// TIA Portal V20 export
FUNCTION_BLOCK "Sequence_1_HotPressLeft"   // FB32858, LAD
TITLE = Sequence
// Sequence template programmend in ladder logic
// stored: IsIECCheckEnabled true, MemoryReserve 100, Namespace Unit1.Em6, SetENOAutomatically true
   VAR_INPUT
      unitStatus { ExternalAccessible := 'False'; ExternalVisible := 'False'; ExternalWritable := 'False'} : "LAF_typeUnitStatus";   // Current unit status o be used in this EM
   END_VAR
   VAR
      instSequenceLADControl { ExternalAccessible := 'False'; ExternalVisible := 'False'; ExternalWritable := 'False'} : "LAF_ControlLadSequence";
      instSequenceLADStatus { ExternalAccessible := 'False'; ExternalVisible := 'False'; ExternalWritable := 'False'} : "LAF_StatusLadSequence";
      statTonTime { ExternalAccessible := 'False'; ExternalVisible := 'False'; ExternalWritable := 'False'} : Array[0..9999] of TON_TIME;
      NoDataCheck { S7_SetPoint := 'True'} : "LER_typePartData";
   END_VAR
   VAR_TEMP
      tempCustomerAction : Bool;   // Placeholder for possible actions
      tempDo_nothing_and_wait_for_init : Bool;   // Placeholder for doing nothing
      tempSafeStateCondition : Bool;   // Temp Condition for the equipment module to be in a safe state
   END_VAR
   VAR CONSTANT
      delayTime : Time := T#500ms;
      STEP_IDLE : DInt := 1;
      JOB_1_STEP_01 : DInt := 101;
      JOB_1_STEP_10 : DInt := 110;
      JOB_1_STEP_20 : DInt := 120;
      JOB_1_STEP_30 : DInt := 130;
      JOB_1_STEP_40 : DInt := 140;
      JOB_1_STEP_41 : DInt := 141;
      JOB_1_STEP_50 : DInt := 150;
      JOB_1_STEP_60 : DInt := 160;
      JOB_1_STEP_70 : DInt := 170;
      JOB_1_STEP_80 : DInt := 180;
      JOB_1_STEP_90 : DInt := 190;
      JOB_2_STEP_01 : DInt := 201;
      JOB_2_STEP_10 : DInt := 210;
      JOB_2_STEP_20 : DInt := 220;
      JOB_2_STEP_30 : DInt := 230;
      JOB_2_STEP_31 : DInt := 231;
      JOB_2_STEP_32 : DInt := 232;
      JOB_2_STEP_40 : DInt := 240;
      JOB_2_STEP_41 : DInt := 241;
      JOB_2_STEP_42 : DInt := 242;
      JOB_2_STEP_43 : DInt := 242;
      JOB_2_STEP_50 : DInt := 250;
      JOB_2_STEP_60 : DInt := 260;
      JOB_2_STEP_70 : DInt := 270;
      JOB_2_STEP_80 : DInt := 280;
      JOB_2_STEP_90 : DInt := 290;
      JOB_3_STEP_01 : DInt := 301;
      JOB_3_STEP_10 : DInt := 310;
      JOB_3_STEP_11 : DInt := 311;
      JOB_3_STEP_20 : DInt := 320;
      JOB_3_STEP_30 : DInt := 330;
      JOB_3_STEP_31 : DInt := 331;
      JOB_3_STEP_32 : DInt := 332;
      JOB_3_STEP_33 : DInt := 333;
      JOB_3_STEP_40 : DInt := 340;
      JOB_3_STEP_41 : DInt := 341;
      JOB_3_STEP_42 : DInt := 342;
      JOB_3_STEP_43 : DInt := 343;
      JOB_3_STEP_50 : DInt := 350;
      JOB_3_STEP_60 : DInt := 360;
      JOB_3_STEP_70 : DInt := 370;
      JOB_3_STEP_80 : DInt := 380;
      JOB_3_STEP_90 : DInt := 390;
      JOB_4_STEP_01 : DInt := 401;
      JOB_4_STEP_10 : DInt := 410;
      JOB_4_STEP_20 : DInt := 420;
      JOB_4_STEP_30 : DInt := 430;
      JOB_4_STEP_31 : DInt := 431;
      JOB_4_STEP_40 : DInt := 440;
      JOB_4_STEP_41 : DInt := 441;
      JOB_4_STEP_42 : DInt := 442;
      JOB_4_STEP_50 : DInt := 450;
      JOB_4_STEP_60 : DInt := 460;
      JOB_4_STEP_70 : DInt := 470;
      JOB_4_STEP_80 : DInt := 480;
      JOB_4_STEP_81 : DInt := 481;
      JOB_4_STEP_90 : DInt := 490;
      JOB_5_STEP_01 : DInt := 501;
      JOB_5_STEP_10 : DInt := 510;
      JOB_5_STEP_11 : DInt := 511;
      JOB_5_STEP_12 : DInt := 512;
      JOB_5_STEP_13 : DInt := 513;
      JOB_5_STEP_20 : DInt := 520;
      JOB_5_STEP_30 : DInt := 530;
      JOB_5_STEP_40 : DInt := 540;
      JOB_5_STEP_41 : DInt := 541;
      JOB_5_STEP_42 : DInt := 542;
      JOB_5_STEP_50 : DInt := 550;
      JOB_5_STEP_60 : DInt := 560;
      JOB_5_STEP_61 : DInt := 561;
      JOB_5_STEP_62 : DInt := 562;
      JOB_5_STEP_63 : DInt := 563;
      JOB_5_STEP_64 : DInt := 564;
      JOB_5_STEP_70 : DInt := 570;
      JOB_5_STEP_80 : DInt := 580;
      JOB_5_STEP_90 : DInt := 590;
      STEP_IMMEDIATE_STOP : DInt := 9001;   // Step executed when an immediate stop command is triggered for the sequence (i.e. when unit is in state aborting)
   END_VAR
   VAR_TEMP   // added for the SCL form of the ladder/FBD networks
      _w1 : Bool;
   END_VAR
BEGIN

REGION Network 1: BLOCK INFO HEADER
   // (company) / (C) Copyright (year)
   // ---------------------------------------------------------------------------------
   // Title:                             (Title of this block)
   // Comment/Function: (that is implemented in the block)
   // Library/Family:           (that the source is dedicated to)
   // Author:                        (department / person in charge / contact)
   // Target System:          (test system with FW version)
   // Engineering:              TIA Portal (SW version)
   // Restrictions:               (OB types, etc.)
   // Requirements:           (hardware, technological package, etc.)
   // ---------------------------------------------------------------------------------
   // Change log table:
   // Version          | Date             | Signature      | Expert in charge  | Changes applied ------------------------|----------------------|-------------------------|--------------------------------|-----------------------
   // 001.000.000 | yyyy-mm-dd | 0x00000000 | (name of expert) | First released version
END_REGION

REGION Network 2: DESCRIPTION
   // This is a template block provided by the Automation Framework. It can be used to create an own project.
   // The Block Info Header is prepared to put in your own data.
   // Description of the block could be added here and the docu created by Code2Docu.
END_REGION

REGION Network 3: ********************* CONTROL *************************
END_REGION

REGION Network 4: Sequence Control ("Enter your Sequins number here")
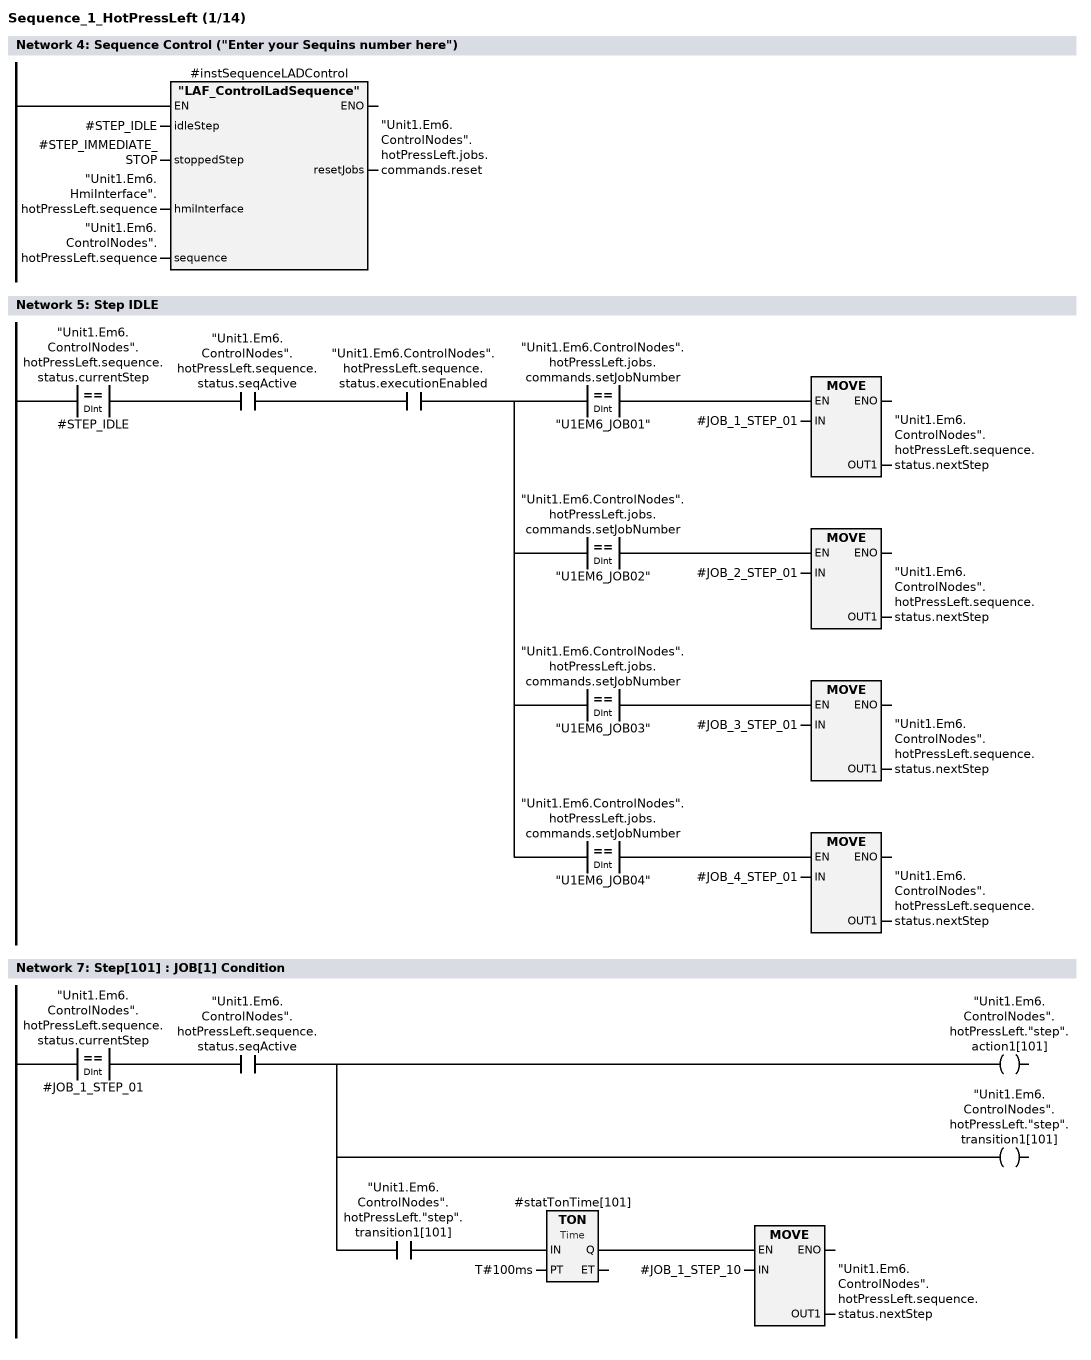
   RUNG wire#powerrail
      #instSequenceLADControl(idleStep := #STEP_IDLE, stoppedStep := #STEP_IMMEDIATE_STOP, hmiInterface := "Unit1.Em6.HmiInterface".hotPressLeft.sequence, sequence := "Unit1.Em6.ControlNodes".hotPressLeft.sequence, resetJobs => "Unit1.Em6.ControlNodes".hotPressLeft.jobs.commands.reset)
   END_RUNG
   // the same network as SCL:
   #instSequenceLADControl(idleStep := #STEP_IDLE,   // "LAF_ControlLadSequence"
                           stoppedStep := #STEP_IMMEDIATE_STOP,
                           hmiInterface := "Unit1.Em6.HmiInterface".hotPressLeft.sequence,
                           sequence := "Unit1.Em6.ControlNodes".hotPressLeft.sequence,
                           resetJobs => "Unit1.Em6.ControlNodes".hotPressLeft.jobs.commands.reset);
END_REGION

REGION Network 5: Step IDLE
   RUNG wire#powerrail
      { S7_Templates := "SrcType := DInt" } EQ_Contact(in1 := "Unit1.Em6.ControlNodes".hotPressLeft.sequence.status.currentStep, in2 := #STEP_IDLE)
      Contact( "Unit1.Em6.ControlNodes".hotPressLeft.sequence.status.seqActive )
      Contact( "Unit1.Em6.ControlNodes".hotPressLeft.sequence.status.executionEnabled )
      wire#w1
      { S7_Templates := "SrcType := DInt" } EQ_Contact(in1 := "Unit1.Em6.ControlNodes".hotPressLeft.jobs.commands.setJobNumber, in2 := "U1EM6_JOB01")
      Move(in := #JOB_1_STEP_01, out1 => "Unit1.Em6.ControlNodes".hotPressLeft.sequence.status.nextStep)
   END_RUNG
   RUNG wire#w1
      { S7_Templates := "SrcType := DInt" } EQ_Contact(in1 := "Unit1.Em6.ControlNodes".hotPressLeft.jobs.commands.setJobNumber, in2 := "U1EM6_JOB02")
      Move(in := #JOB_2_STEP_01, out1 => "Unit1.Em6.ControlNodes".hotPressLeft.sequence.status.nextStep)
   END_RUNG
   RUNG wire#w1
      { S7_Templates := "SrcType := DInt" } EQ_Contact(in1 := "Unit1.Em6.ControlNodes".hotPressLeft.jobs.commands.setJobNumber, in2 := "U1EM6_JOB03")
      Move(in := #JOB_3_STEP_01, out1 => "Unit1.Em6.ControlNodes".hotPressLeft.sequence.status.nextStep)
   END_RUNG
   RUNG wire#w1
      { S7_Templates := "SrcType := DInt" } EQ_Contact(in1 := "Unit1.Em6.ControlNodes".hotPressLeft.jobs.commands.setJobNumber, in2 := "U1EM6_JOB04")
      Move(in := #JOB_4_STEP_01, out1 => "Unit1.Em6.ControlNodes".hotPressLeft.sequence.status.nextStep)
   END_RUNG
   // the same network as SCL:
   #_w1 := ("Unit1.Em6.ControlNodes".hotPressLeft.sequence.status.currentStep = #STEP_IDLE) AND "Unit1.Em6.ControlNodes".hotPressLeft.sequence.status.seqActive AND "Unit1.Em6.ControlNodes".hotPressLeft.sequence.status.executionEnabled;
   IF #_w1 AND ("Unit1.Em6.ControlNodes".hotPressLeft.jobs.commands.setJobNumber = "U1EM6_JOB01") THEN
       "Unit1.Em6.ControlNodes".hotPressLeft.sequence.status.nextStep := #JOB_1_STEP_01;
   END_IF;
   IF #_w1 AND ("Unit1.Em6.ControlNodes".hotPressLeft.jobs.commands.setJobNumber = "U1EM6_JOB02") THEN
       "Unit1.Em6.ControlNodes".hotPressLeft.sequence.status.nextStep := #JOB_2_STEP_01;
   END_IF;
   IF #_w1 AND ("Unit1.Em6.ControlNodes".hotPressLeft.jobs.commands.setJobNumber = "U1EM6_JOB03") THEN
       "Unit1.Em6.ControlNodes".hotPressLeft.sequence.status.nextStep := #JOB_3_STEP_01;
   END_IF;
   IF #_w1 AND ("Unit1.Em6.ControlNodes".hotPressLeft.jobs.commands.setJobNumber = "U1EM6_JOB04") THEN
       "Unit1.Em6.ControlNodes".hotPressLeft.sequence.status.nextStep := #JOB_4_STEP_01;
   END_IF;
END_REGION

REGION Network 6: *************** JOB[1] EM HOMING ************************
END_REGION

REGION Network 7: Step[101] : JOB[1] Condition
   RUNG wire#powerrail
      { S7_Templates := "SrcType := DInt" } EQ_Contact(in1 := "Unit1.Em6.ControlNodes".hotPressLeft.sequence.status.currentStep, in2 := #JOB_1_STEP_01)
      Contact( "Unit1.Em6.ControlNodes".hotPressLeft.sequence.status.seqActive )
      wire#w1
      Coil( "Unit1.Em6.ControlNodes".hotPressLeft."step".action1[101] )
   END_RUNG
   RUNG wire#w1
      Coil( "Unit1.Em6.ControlNodes".hotPressLeft."step".transition1[101] )
   END_RUNG
   RUNG wire#w1
      Contact( "Unit1.Em6.ControlNodes".hotPressLeft."step".transition1[101] )
      { S7_Templates := "time_type := Time" } #statTonTime[101].TON(pt := T#100ms, et =>)
      Move(in := #JOB_1_STEP_10, out1 => "Unit1.Em6.ControlNodes".hotPressLeft.sequence.status.nextStep)
   END_RUNG
   // the same network as SCL:
   "Unit1.Em6.ControlNodes".hotPressLeft."step".action1[101] := ("Unit1.Em6.ControlNodes".hotPressLeft.sequence.status.currentStep = #JOB_1_STEP_01) AND "Unit1.Em6.ControlNodes".hotPressLeft.sequence.status.seqActive;
   "Unit1.Em6.ControlNodes".hotPressLeft."step".transition1[101] := ("Unit1.Em6.ControlNodes".hotPressLeft.sequence.status.currentStep = #JOB_1_STEP_01) AND "Unit1.Em6.ControlNodes".hotPressLeft.sequence.status.seqActive;
   #statTonTime[101].TON(IN := ("Unit1.Em6.ControlNodes".hotPressLeft.sequence.status.currentStep = #JOB_1_STEP_01) AND "Unit1.Em6.ControlNodes".hotPressLeft.sequence.status.seqActive AND "Unit1.Em6.ControlNodes".hotPressLeft."step".transition1[101],
                         PT := T#100ms);
   IF #statTonTime[101].Q THEN
       "Unit1.Em6.ControlNodes".hotPressLeft.sequence.status.nextStep := #JOB_1_STEP_10;
   END_IF;
END_REGION

REGION Network 8: Step[110] : Servo Press Reference Home Pos
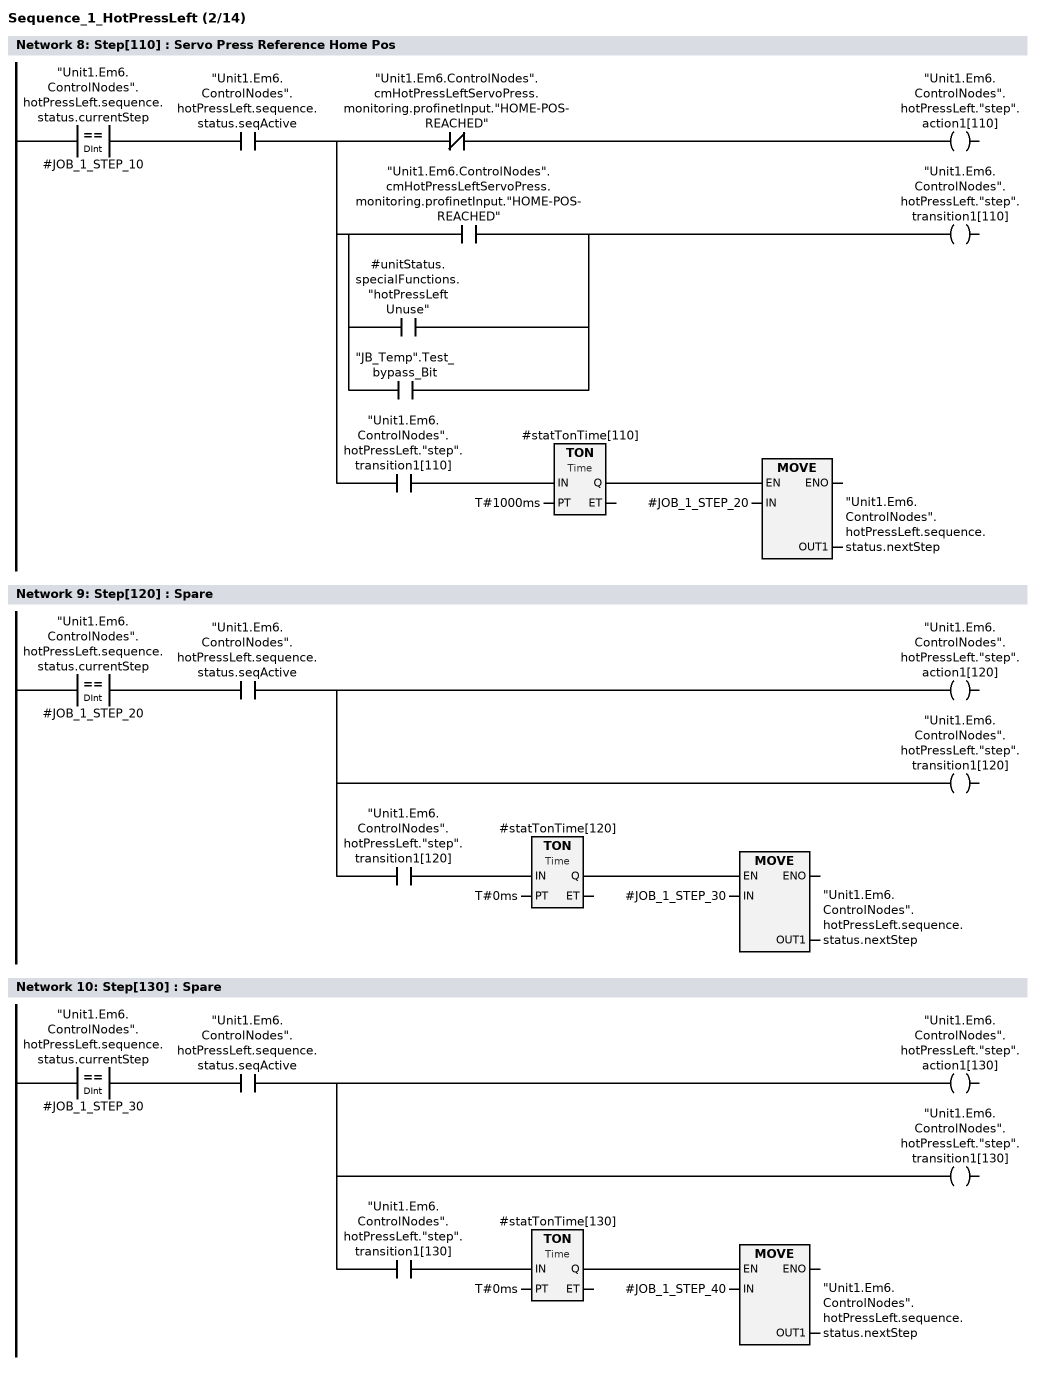
   RUNG wire#powerrail
      { S7_Templates := "SrcType := DInt" } EQ_Contact(in1 := "Unit1.Em6.ControlNodes".hotPressLeft.sequence.status.currentStep, in2 := #JOB_1_STEP_10)
      Contact( "Unit1.Em6.ControlNodes".hotPressLeft.sequence.status.seqActive )
      wire#w1
      I_Contact( "Unit1.Em6.ControlNodes".cmHotPressLeftServoPress.monitoring.profinetInput."HOME-POS-REACHED" )
      Coil( "Unit1.Em6.ControlNodes".hotPressLeft."step".action1[110] )
   END_RUNG
   RUNG wire#w1
      Contact( "Unit1.Em6.ControlNodes".cmHotPressLeftServoPress.monitoring.profinetInput."HOME-POS-REACHED" )
      wire#w2
      Coil( "Unit1.Em6.ControlNodes".hotPressLeft."step".transition1[110] )
   END_RUNG
   RUNG wire#w1
      Contact( #unitStatus.specialFunctions."hotPressLeft Unuse" )
   END_RUNG wire#w2
   RUNG wire#w1
      Contact( "JB_Temp".Test_bypass_Bit )
   END_RUNG wire#w2
   RUNG wire#w1
      Contact( "Unit1.Em6.ControlNodes".hotPressLeft."step".transition1[110] )
      { S7_Templates := "time_type := Time" } #statTonTime[110].TON(pt := T#1000ms, et =>)
      Move(in := #JOB_1_STEP_20, out1 => "Unit1.Em6.ControlNodes".hotPressLeft.sequence.status.nextStep)
   END_RUNG
   // the same network as SCL:
   #_w1 := ("Unit1.Em6.ControlNodes".hotPressLeft.sequence.status.currentStep = #JOB_1_STEP_10) AND "Unit1.Em6.ControlNodes".hotPressLeft.sequence.status.seqActive;
   "Unit1.Em6.ControlNodes".hotPressLeft."step".action1[110] := #_w1 AND NOT "Unit1.Em6.ControlNodes".cmHotPressLeftServoPress.monitoring.profinetInput."HOME-POS-REACHED";
   "Unit1.Em6.ControlNodes".hotPressLeft."step".transition1[110] := #_w1 AND ("Unit1.Em6.ControlNodes".cmHotPressLeftServoPress.monitoring.profinetInput."HOME-POS-REACHED" OR #unitStatus.specialFunctions."hotPressLeft Unuse" OR "JB_Temp".Test_bypass_Bit);
   #statTonTime[110].TON(IN := #_w1 AND "Unit1.Em6.ControlNodes".hotPressLeft."step".transition1[110],
                         PT := T#1000ms);
   IF #statTonTime[110].Q THEN
       "Unit1.Em6.ControlNodes".hotPressLeft.sequence.status.nextStep := #JOB_1_STEP_20;
   END_IF;
END_REGION

REGION Network 9: Step[120] : Spare
   RUNG wire#powerrail
      { S7_Templates := "SrcType := DInt" } EQ_Contact(in1 := "Unit1.Em6.ControlNodes".hotPressLeft.sequence.status.currentStep, in2 := #JOB_1_STEP_20)
      Contact( "Unit1.Em6.ControlNodes".hotPressLeft.sequence.status.seqActive )
      wire#w1
      Coil( "Unit1.Em6.ControlNodes".hotPressLeft."step".action1[120] )
   END_RUNG
   RUNG wire#w1
      Coil( "Unit1.Em6.ControlNodes".hotPressLeft."step".transition1[120] )
   END_RUNG
   RUNG wire#w1
      Contact( "Unit1.Em6.ControlNodes".hotPressLeft."step".transition1[120] )
      { S7_Templates := "time_type := Time" } #statTonTime[120].TON(pt := T#0ms, et =>)
      Move(in := #JOB_1_STEP_30, out1 => "Unit1.Em6.ControlNodes".hotPressLeft.sequence.status.nextStep)
   END_RUNG
   // the same network as SCL:
   "Unit1.Em6.ControlNodes".hotPressLeft."step".action1[120] := ("Unit1.Em6.ControlNodes".hotPressLeft.sequence.status.currentStep = #JOB_1_STEP_20) AND "Unit1.Em6.ControlNodes".hotPressLeft.sequence.status.seqActive;
   "Unit1.Em6.ControlNodes".hotPressLeft."step".transition1[120] := ("Unit1.Em6.ControlNodes".hotPressLeft.sequence.status.currentStep = #JOB_1_STEP_20) AND "Unit1.Em6.ControlNodes".hotPressLeft.sequence.status.seqActive;
   #statTonTime[120].TON(IN := ("Unit1.Em6.ControlNodes".hotPressLeft.sequence.status.currentStep = #JOB_1_STEP_20) AND "Unit1.Em6.ControlNodes".hotPressLeft.sequence.status.seqActive AND "Unit1.Em6.ControlNodes".hotPressLeft."step".transition1[120],
                         PT := T#0ms);
   IF #statTonTime[120].Q THEN
       "Unit1.Em6.ControlNodes".hotPressLeft.sequence.status.nextStep := #JOB_1_STEP_30;
   END_IF;
END_REGION

REGION Network 10: Step[130] : Spare
   RUNG wire#powerrail
      { S7_Templates := "SrcType := DInt" } EQ_Contact(in1 := "Unit1.Em6.ControlNodes".hotPressLeft.sequence.status.currentStep, in2 := #JOB_1_STEP_30)
      Contact( "Unit1.Em6.ControlNodes".hotPressLeft.sequence.status.seqActive )
      wire#w1
      Coil( "Unit1.Em6.ControlNodes".hotPressLeft."step".action1[130] )
   END_RUNG
   RUNG wire#w1
      Coil( "Unit1.Em6.ControlNodes".hotPressLeft."step".transition1[130] )
   END_RUNG
   RUNG wire#w1
      Contact( "Unit1.Em6.ControlNodes".hotPressLeft."step".transition1[130] )
      { S7_Templates := "time_type := Time" } #statTonTime[130].TON(pt := T#0ms, et =>)
      Move(in := #JOB_1_STEP_40, out1 => "Unit1.Em6.ControlNodes".hotPressLeft.sequence.status.nextStep)
   END_RUNG
   // the same network as SCL:
   "Unit1.Em6.ControlNodes".hotPressLeft."step".action1[130] := ("Unit1.Em6.ControlNodes".hotPressLeft.sequence.status.currentStep = #JOB_1_STEP_30) AND "Unit1.Em6.ControlNodes".hotPressLeft.sequence.status.seqActive;
   "Unit1.Em6.ControlNodes".hotPressLeft."step".transition1[130] := ("Unit1.Em6.ControlNodes".hotPressLeft.sequence.status.currentStep = #JOB_1_STEP_30) AND "Unit1.Em6.ControlNodes".hotPressLeft.sequence.status.seqActive;
   #statTonTime[130].TON(IN := ("Unit1.Em6.ControlNodes".hotPressLeft.sequence.status.currentStep = #JOB_1_STEP_30) AND "Unit1.Em6.ControlNodes".hotPressLeft.sequence.status.seqActive AND "Unit1.Em6.ControlNodes".hotPressLeft."step".transition1[130],
                         PT := T#0ms);
   IF #statTonTime[130].Q THEN
       "Unit1.Em6.ControlNodes".hotPressLeft.sequence.status.nextStep := #JOB_1_STEP_40;
   END_IF;
END_REGION

REGION Network 11: Step[140] : Spare
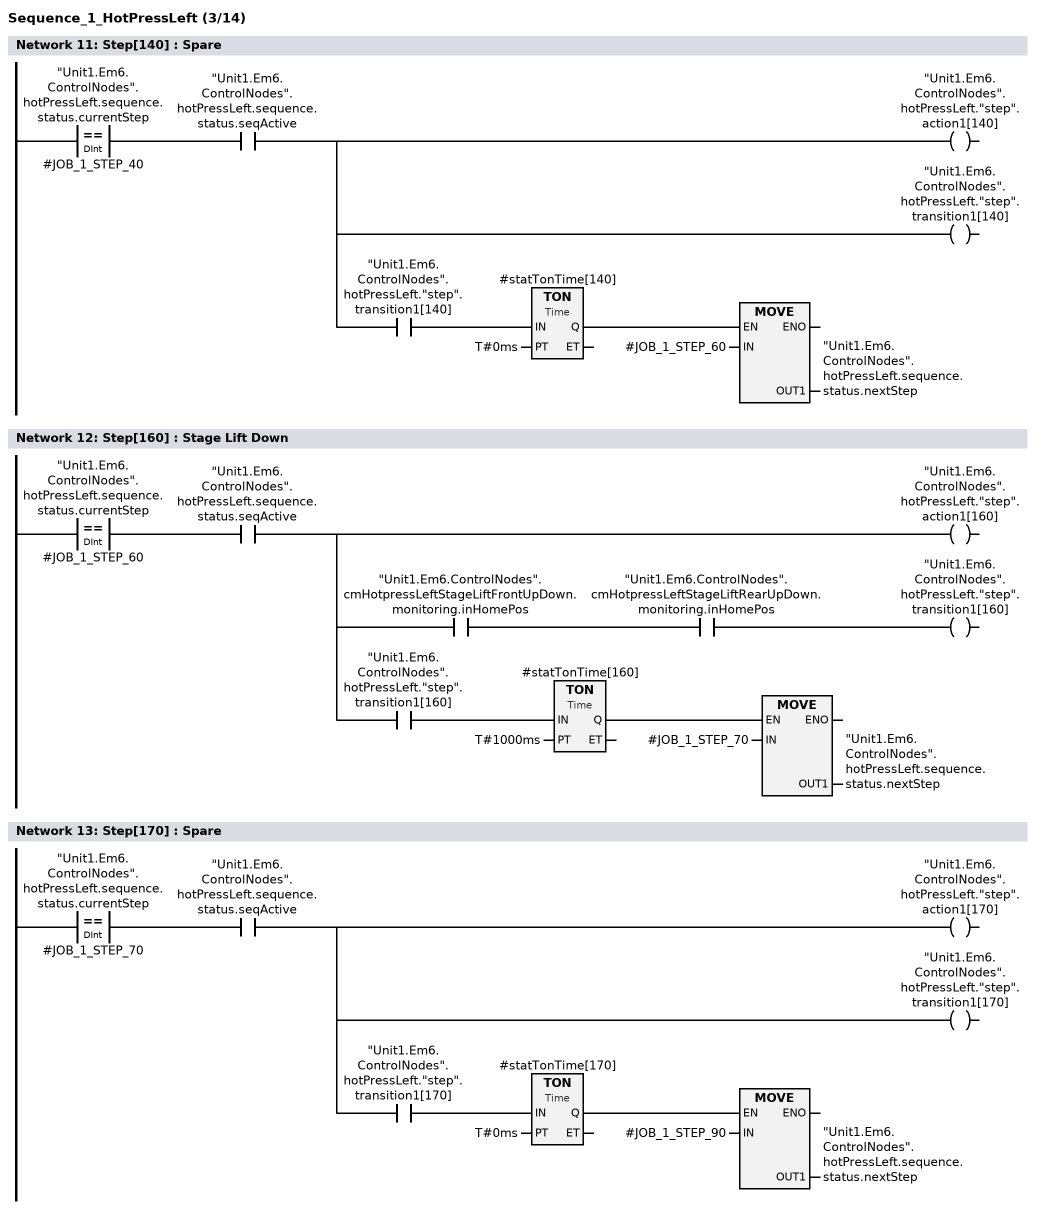
   RUNG wire#powerrail
      { S7_Templates := "SrcType := DInt" } EQ_Contact(in1 := "Unit1.Em6.ControlNodes".hotPressLeft.sequence.status.currentStep, in2 := #JOB_1_STEP_40)
      Contact( "Unit1.Em6.ControlNodes".hotPressLeft.sequence.status.seqActive )
      wire#w1
      Coil( "Unit1.Em6.ControlNodes".hotPressLeft."step".action1[140] )
   END_RUNG
   RUNG wire#w1
      Coil( "Unit1.Em6.ControlNodes".hotPressLeft."step".transition1[140] )
   END_RUNG
   RUNG wire#w1
      Contact( "Unit1.Em6.ControlNodes".hotPressLeft."step".transition1[140] )
      { S7_Templates := "time_type := Time" } #statTonTime[140].TON(pt := T#0ms, et =>)
      Move(in := #JOB_1_STEP_60, out1 => "Unit1.Em6.ControlNodes".hotPressLeft.sequence.status.nextStep)
   END_RUNG
   // the same network as SCL:
   "Unit1.Em6.ControlNodes".hotPressLeft."step".action1[140] := ("Unit1.Em6.ControlNodes".hotPressLeft.sequence.status.currentStep = #JOB_1_STEP_40) AND "Unit1.Em6.ControlNodes".hotPressLeft.sequence.status.seqActive;
   "Unit1.Em6.ControlNodes".hotPressLeft."step".transition1[140] := ("Unit1.Em6.ControlNodes".hotPressLeft.sequence.status.currentStep = #JOB_1_STEP_40) AND "Unit1.Em6.ControlNodes".hotPressLeft.sequence.status.seqActive;
   #statTonTime[140].TON(IN := ("Unit1.Em6.ControlNodes".hotPressLeft.sequence.status.currentStep = #JOB_1_STEP_40) AND "Unit1.Em6.ControlNodes".hotPressLeft.sequence.status.seqActive AND "Unit1.Em6.ControlNodes".hotPressLeft."step".transition1[140],
                         PT := T#0ms);
   IF #statTonTime[140].Q THEN
       "Unit1.Em6.ControlNodes".hotPressLeft.sequence.status.nextStep := #JOB_1_STEP_60;
   END_IF;
END_REGION

REGION Network 12: Step[160] : Stage Lift Down
   RUNG wire#powerrail
      { S7_Templates := "SrcType := DInt" } EQ_Contact(in1 := "Unit1.Em6.ControlNodes".hotPressLeft.sequence.status.currentStep, in2 := #JOB_1_STEP_60)
      Contact( "Unit1.Em6.ControlNodes".hotPressLeft.sequence.status.seqActive )
      wire#w1
      Coil( "Unit1.Em6.ControlNodes".hotPressLeft."step".action1[160] )
   END_RUNG
   RUNG wire#w1
      Contact( "Unit1.Em6.ControlNodes".cmHotpressLeftStageLiftFrontUpDown.monitoring.inHomePos )
      Contact( "Unit1.Em6.ControlNodes".cmHotpressLeftStageLiftRearUpDown.monitoring.inHomePos )
      Coil( "Unit1.Em6.ControlNodes".hotPressLeft."step".transition1[160] )
   END_RUNG
   RUNG wire#w1
      Contact( "Unit1.Em6.ControlNodes".hotPressLeft."step".transition1[160] )
      { S7_Templates := "time_type := Time" } #statTonTime[160].TON(pt := T#1000ms, et =>)
      Move(in := #JOB_1_STEP_70, out1 => "Unit1.Em6.ControlNodes".hotPressLeft.sequence.status.nextStep)
   END_RUNG
   // the same network as SCL:
   "Unit1.Em6.ControlNodes".hotPressLeft."step".action1[160] := ("Unit1.Em6.ControlNodes".hotPressLeft.sequence.status.currentStep = #JOB_1_STEP_60) AND "Unit1.Em6.ControlNodes".hotPressLeft.sequence.status.seqActive;
   "Unit1.Em6.ControlNodes".hotPressLeft."step".transition1[160] := ("Unit1.Em6.ControlNodes".hotPressLeft.sequence.status.currentStep = #JOB_1_STEP_60) AND "Unit1.Em6.ControlNodes".hotPressLeft.sequence.status.seqActive AND "Unit1.Em6.ControlNodes".cmHotpressLeftStageLiftFrontUpDown.monitoring.inHomePos AND "Unit1.Em6.ControlNodes".cmHotpressLeftStageLiftRearUpDown.monitoring.inHomePos;
   #statTonTime[160].TON(IN := ("Unit1.Em6.ControlNodes".hotPressLeft.sequence.status.currentStep = #JOB_1_STEP_60) AND "Unit1.Em6.ControlNodes".hotPressLeft.sequence.status.seqActive AND "Unit1.Em6.ControlNodes".hotPressLeft."step".transition1[160],
                         PT := T#1000ms);
   IF #statTonTime[160].Q THEN
       "Unit1.Em6.ControlNodes".hotPressLeft.sequence.status.nextStep := #JOB_1_STEP_70;
   END_IF;
END_REGION

REGION Network 13: Step[170] : Spare
   RUNG wire#powerrail
      { S7_Templates := "SrcType := DInt" } EQ_Contact(in1 := "Unit1.Em6.ControlNodes".hotPressLeft.sequence.status.currentStep, in2 := #JOB_1_STEP_70)
      Contact( "Unit1.Em6.ControlNodes".hotPressLeft.sequence.status.seqActive )
      wire#w1
      Coil( "Unit1.Em6.ControlNodes".hotPressLeft."step".action1[170] )
   END_RUNG
   RUNG wire#w1
      Coil( "Unit1.Em6.ControlNodes".hotPressLeft."step".transition1[170] )
   END_RUNG
   RUNG wire#w1
      Contact( "Unit1.Em6.ControlNodes".hotPressLeft."step".transition1[170] )
      { S7_Templates := "time_type := Time" } #statTonTime[170].TON(pt := T#0ms, et =>)
      Move(in := #JOB_1_STEP_90, out1 => "Unit1.Em6.ControlNodes".hotPressLeft.sequence.status.nextStep)
   END_RUNG
   // the same network as SCL:
   "Unit1.Em6.ControlNodes".hotPressLeft."step".action1[170] := ("Unit1.Em6.ControlNodes".hotPressLeft.sequence.status.currentStep = #JOB_1_STEP_70) AND "Unit1.Em6.ControlNodes".hotPressLeft.sequence.status.seqActive;
   "Unit1.Em6.ControlNodes".hotPressLeft."step".transition1[170] := ("Unit1.Em6.ControlNodes".hotPressLeft.sequence.status.currentStep = #JOB_1_STEP_70) AND "Unit1.Em6.ControlNodes".hotPressLeft.sequence.status.seqActive;
   #statTonTime[170].TON(IN := ("Unit1.Em6.ControlNodes".hotPressLeft.sequence.status.currentStep = #JOB_1_STEP_70) AND "Unit1.Em6.ControlNodes".hotPressLeft.sequence.status.seqActive AND "Unit1.Em6.ControlNodes".hotPressLeft."step".transition1[170],
                         PT := T#0ms);
   IF #statTonTime[170].Q THEN
       "Unit1.Em6.ControlNodes".hotPressLeft.sequence.status.nextStep := #JOB_1_STEP_90;
   END_IF;
END_REGION

REGION Network 14: Step[190] : JOB[1] Step End
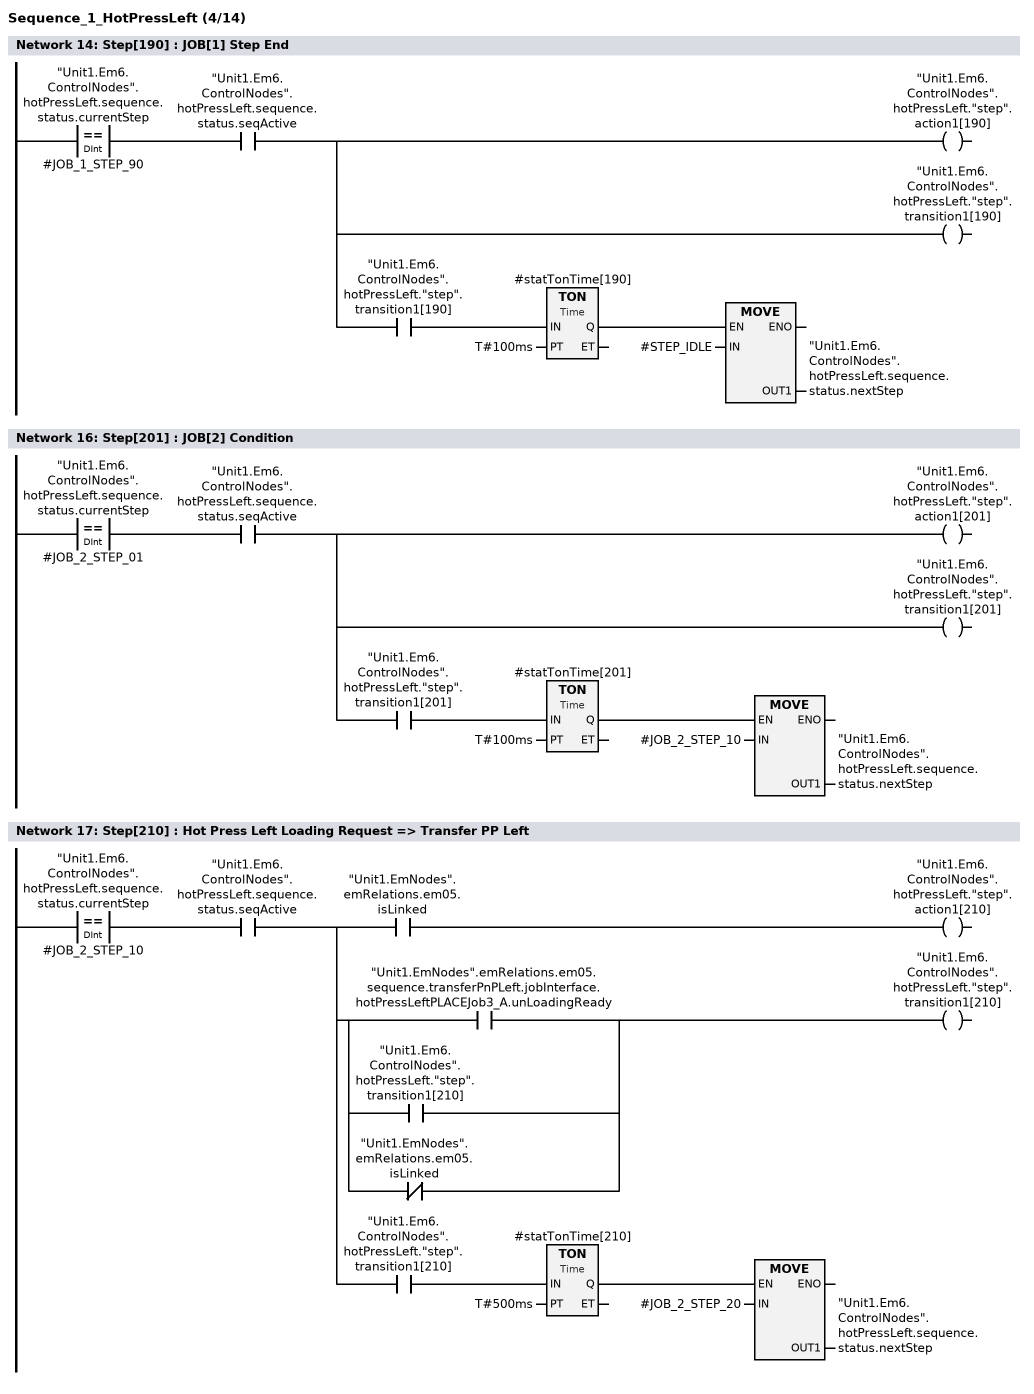
   RUNG wire#powerrail
      { S7_Templates := "SrcType := DInt" } EQ_Contact(in1 := "Unit1.Em6.ControlNodes".hotPressLeft.sequence.status.currentStep, in2 := #JOB_1_STEP_90)
      Contact( "Unit1.Em6.ControlNodes".hotPressLeft.sequence.status.seqActive )
      wire#w1
      Coil( "Unit1.Em6.ControlNodes".hotPressLeft."step".action1[190] )
   END_RUNG
   RUNG wire#w1
      Coil( "Unit1.Em6.ControlNodes".hotPressLeft."step".transition1[190] )
   END_RUNG
   RUNG wire#w1
      Contact( "Unit1.Em6.ControlNodes".hotPressLeft."step".transition1[190] )
      { S7_Templates := "time_type := Time" } #statTonTime[190].TON(pt := T#100ms, et =>)
      Move(in := #STEP_IDLE, out1 => "Unit1.Em6.ControlNodes".hotPressLeft.sequence.status.nextStep)
   END_RUNG
   // the same network as SCL:
   "Unit1.Em6.ControlNodes".hotPressLeft."step".action1[190] := ("Unit1.Em6.ControlNodes".hotPressLeft.sequence.status.currentStep = #JOB_1_STEP_90) AND "Unit1.Em6.ControlNodes".hotPressLeft.sequence.status.seqActive;
   "Unit1.Em6.ControlNodes".hotPressLeft."step".transition1[190] := ("Unit1.Em6.ControlNodes".hotPressLeft.sequence.status.currentStep = #JOB_1_STEP_90) AND "Unit1.Em6.ControlNodes".hotPressLeft.sequence.status.seqActive;
   #statTonTime[190].TON(IN := ("Unit1.Em6.ControlNodes".hotPressLeft.sequence.status.currentStep = #JOB_1_STEP_90) AND "Unit1.Em6.ControlNodes".hotPressLeft.sequence.status.seqActive AND "Unit1.Em6.ControlNodes".hotPressLeft."step".transition1[190],
                         PT := T#100ms);
   IF #statTonTime[190].Q THEN
       "Unit1.Em6.ControlNodes".hotPressLeft.sequence.status.nextStep := #STEP_IDLE;
   END_IF;
END_REGION

REGION Network 15: *************** JOB[2] JR GET=AUTO **********************
END_REGION

REGION Network 16: Step[201] : JOB[2] Condition
   RUNG wire#powerrail
      { S7_Templates := "SrcType := DInt" } EQ_Contact(in1 := "Unit1.Em6.ControlNodes".hotPressLeft.sequence.status.currentStep, in2 := #JOB_2_STEP_01)
      Contact( "Unit1.Em6.ControlNodes".hotPressLeft.sequence.status.seqActive )
      wire#w1
      Coil( "Unit1.Em6.ControlNodes".hotPressLeft."step".action1[201] )
   END_RUNG
   RUNG wire#w1
      Coil( "Unit1.Em6.ControlNodes".hotPressLeft."step".transition1[201] )
   END_RUNG
   RUNG wire#w1
      Contact( "Unit1.Em6.ControlNodes".hotPressLeft."step".transition1[201] )
      { S7_Templates := "time_type := Time" } #statTonTime[201].TON(pt := T#100ms, et =>)
      Move(in := #JOB_2_STEP_10, out1 => "Unit1.Em6.ControlNodes".hotPressLeft.sequence.status.nextStep)
   END_RUNG
   // the same network as SCL:
   "Unit1.Em6.ControlNodes".hotPressLeft."step".action1[201] := ("Unit1.Em6.ControlNodes".hotPressLeft.sequence.status.currentStep = #JOB_2_STEP_01) AND "Unit1.Em6.ControlNodes".hotPressLeft.sequence.status.seqActive;
   "Unit1.Em6.ControlNodes".hotPressLeft."step".transition1[201] := ("Unit1.Em6.ControlNodes".hotPressLeft.sequence.status.currentStep = #JOB_2_STEP_01) AND "Unit1.Em6.ControlNodes".hotPressLeft.sequence.status.seqActive;
   #statTonTime[201].TON(IN := ("Unit1.Em6.ControlNodes".hotPressLeft.sequence.status.currentStep = #JOB_2_STEP_01) AND "Unit1.Em6.ControlNodes".hotPressLeft.sequence.status.seqActive AND "Unit1.Em6.ControlNodes".hotPressLeft."step".transition1[201],
                         PT := T#100ms);
   IF #statTonTime[201].Q THEN
       "Unit1.Em6.ControlNodes".hotPressLeft.sequence.status.nextStep := #JOB_2_STEP_10;
   END_IF;
END_REGION

REGION Network 17: Step[210] : Hot Press Left Loading Request => Transfer PP Left
   RUNG wire#powerrail
      { S7_Templates := "SrcType := DInt" } EQ_Contact(in1 := "Unit1.Em6.ControlNodes".hotPressLeft.sequence.status.currentStep, in2 := #JOB_2_STEP_10)
      Contact( "Unit1.Em6.ControlNodes".hotPressLeft.sequence.status.seqActive )
      wire#w1
      Contact( "Unit1.EmNodes".emRelations.em05.isLinked )
      Coil( "Unit1.Em6.ControlNodes".hotPressLeft."step".action1[210] )
   END_RUNG
   RUNG wire#w1
      Contact( "Unit1.EmNodes".emRelations.em05.sequence.transferPnPLeft.jobInterface.hotPressLeftPLACEJob3_A.unLoadingReady )
      wire#w2
      Coil( "Unit1.Em6.ControlNodes".hotPressLeft."step".transition1[210] )
   END_RUNG
   RUNG wire#w1
      Contact( "Unit1.Em6.ControlNodes".hotPressLeft."step".transition1[210] )
   END_RUNG wire#w2
   RUNG wire#w1
      I_Contact( "Unit1.EmNodes".emRelations.em05.isLinked )
   END_RUNG wire#w2
   RUNG wire#w1
      Contact( "Unit1.Em6.ControlNodes".hotPressLeft."step".transition1[210] )
      { S7_Templates := "time_type := Time" } #statTonTime[210].TON(pt := T#500ms, et =>)
      Move(in := #JOB_2_STEP_20, out1 => "Unit1.Em6.ControlNodes".hotPressLeft.sequence.status.nextStep)
   END_RUNG
   // the same network as SCL:
   #_w1 := ("Unit1.Em6.ControlNodes".hotPressLeft.sequence.status.currentStep = #JOB_2_STEP_10) AND "Unit1.Em6.ControlNodes".hotPressLeft.sequence.status.seqActive;
   "Unit1.Em6.ControlNodes".hotPressLeft."step".action1[210] := #_w1 AND "Unit1.EmNodes".emRelations.em05.isLinked;
   "Unit1.Em6.ControlNodes".hotPressLeft."step".transition1[210] := #_w1 AND ("Unit1.EmNodes".emRelations.em05.sequence.transferPnPLeft.jobInterface.hotPressLeftPLACEJob3_A.unLoadingReady OR "Unit1.Em6.ControlNodes".hotPressLeft."step".transition1[210] OR NOT "Unit1.EmNodes".emRelations.em05.isLinked);
   #statTonTime[210].TON(IN := #_w1 AND "Unit1.Em6.ControlNodes".hotPressLeft."step".transition1[210],
                         PT := T#500ms);
   IF #statTonTime[210].Q THEN
       "Unit1.Em6.ControlNodes".hotPressLeft.sequence.status.nextStep := #JOB_2_STEP_20;
   END_IF;
END_REGION

REGION Network 18: Step[220] : Spare
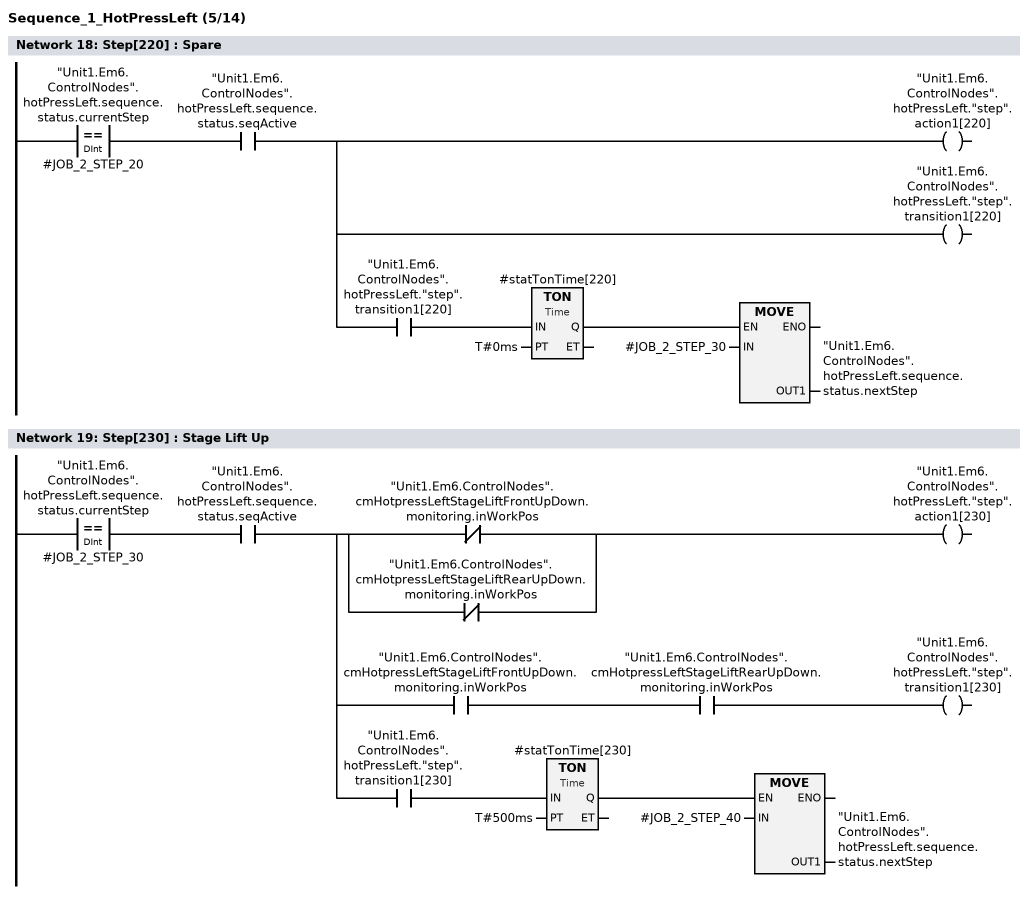
   RUNG wire#powerrail
      { S7_Templates := "SrcType := DInt" } EQ_Contact(in1 := "Unit1.Em6.ControlNodes".hotPressLeft.sequence.status.currentStep, in2 := #JOB_2_STEP_20)
      Contact( "Unit1.Em6.ControlNodes".hotPressLeft.sequence.status.seqActive )
      wire#w1
      Coil( "Unit1.Em6.ControlNodes".hotPressLeft."step".action1[220] )
   END_RUNG
   RUNG wire#w1
      Coil( "Unit1.Em6.ControlNodes".hotPressLeft."step".transition1[220] )
   END_RUNG
   RUNG wire#w1
      Contact( "Unit1.Em6.ControlNodes".hotPressLeft."step".transition1[220] )
      { S7_Templates := "time_type := Time" } #statTonTime[220].TON(pt := T#0ms, et =>)
      Move(in := #JOB_2_STEP_30, out1 => "Unit1.Em6.ControlNodes".hotPressLeft.sequence.status.nextStep)
   END_RUNG
   // the same network as SCL:
   "Unit1.Em6.ControlNodes".hotPressLeft."step".action1[220] := ("Unit1.Em6.ControlNodes".hotPressLeft.sequence.status.currentStep = #JOB_2_STEP_20) AND "Unit1.Em6.ControlNodes".hotPressLeft.sequence.status.seqActive;
   "Unit1.Em6.ControlNodes".hotPressLeft."step".transition1[220] := ("Unit1.Em6.ControlNodes".hotPressLeft.sequence.status.currentStep = #JOB_2_STEP_20) AND "Unit1.Em6.ControlNodes".hotPressLeft.sequence.status.seqActive;
   #statTonTime[220].TON(IN := ("Unit1.Em6.ControlNodes".hotPressLeft.sequence.status.currentStep = #JOB_2_STEP_20) AND "Unit1.Em6.ControlNodes".hotPressLeft.sequence.status.seqActive AND "Unit1.Em6.ControlNodes".hotPressLeft."step".transition1[220],
                         PT := T#0ms);
   IF #statTonTime[220].Q THEN
       "Unit1.Em6.ControlNodes".hotPressLeft.sequence.status.nextStep := #JOB_2_STEP_30;
   END_IF;
END_REGION

REGION Network 19: Step[230] : Stage Lift Up
   RUNG wire#powerrail
      { S7_Templates := "SrcType := DInt" } EQ_Contact(in1 := "Unit1.Em6.ControlNodes".hotPressLeft.sequence.status.currentStep, in2 := #JOB_2_STEP_30)
      Contact( "Unit1.Em6.ControlNodes".hotPressLeft.sequence.status.seqActive )
      wire#w1
      I_Contact( "Unit1.Em6.ControlNodes".cmHotpressLeftStageLiftFrontUpDown.monitoring.inWorkPos )
      wire#w2
      Coil( "Unit1.Em6.ControlNodes".hotPressLeft."step".action1[230] )
   END_RUNG
   RUNG wire#w1
      I_Contact( "Unit1.Em6.ControlNodes".cmHotpressLeftStageLiftRearUpDown.monitoring.inWorkPos )
   END_RUNG wire#w2
   RUNG wire#w1
      Contact( "Unit1.Em6.ControlNodes".cmHotpressLeftStageLiftFrontUpDown.monitoring.inWorkPos )
      Contact( "Unit1.Em6.ControlNodes".cmHotpressLeftStageLiftRearUpDown.monitoring.inWorkPos )
      Coil( "Unit1.Em6.ControlNodes".hotPressLeft."step".transition1[230] )
   END_RUNG
   RUNG wire#w1
      Contact( "Unit1.Em6.ControlNodes".hotPressLeft."step".transition1[230] )
      { S7_Templates := "time_type := Time" } #statTonTime[230].TON(pt := T#500ms, et =>)
      Move(in := #JOB_2_STEP_40, out1 => "Unit1.Em6.ControlNodes".hotPressLeft.sequence.status.nextStep)
   END_RUNG
   // the same network as SCL:
   #_w1 := ("Unit1.Em6.ControlNodes".hotPressLeft.sequence.status.currentStep = #JOB_2_STEP_30) AND "Unit1.Em6.ControlNodes".hotPressLeft.sequence.status.seqActive;
   "Unit1.Em6.ControlNodes".hotPressLeft."step".action1[230] := #_w1 AND (NOT "Unit1.Em6.ControlNodes".cmHotpressLeftStageLiftFrontUpDown.monitoring.inWorkPos OR NOT "Unit1.Em6.ControlNodes".cmHotpressLeftStageLiftRearUpDown.monitoring.inWorkPos);
   "Unit1.Em6.ControlNodes".hotPressLeft."step".transition1[230] := #_w1 AND "Unit1.Em6.ControlNodes".cmHotpressLeftStageLiftFrontUpDown.monitoring.inWorkPos AND "Unit1.Em6.ControlNodes".cmHotpressLeftStageLiftRearUpDown.monitoring.inWorkPos;
   #statTonTime[230].TON(IN := #_w1 AND "Unit1.Em6.ControlNodes".hotPressLeft."step".transition1[230],
                         PT := T#500ms);
   IF #statTonTime[230].Q THEN
       "Unit1.Em6.ControlNodes".hotPressLeft.sequence.status.nextStep := #JOB_2_STEP_40;
   END_IF;
END_REGION

REGION Network 20: Step[240] : Hot Press Left Loading Check => Transfer PP Left
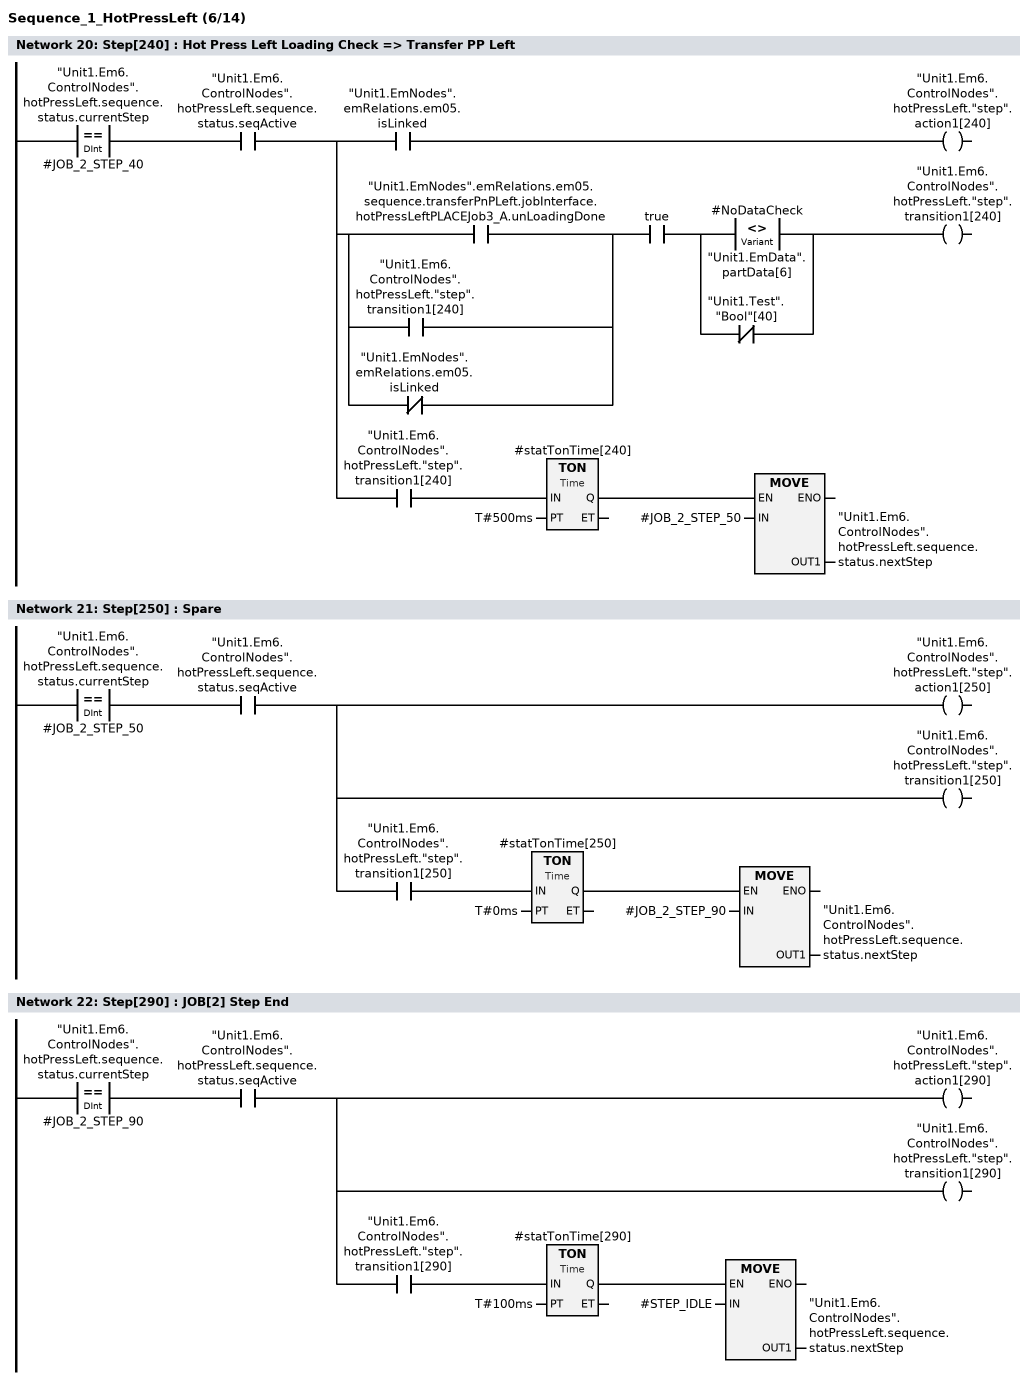
   RUNG wire#powerrail
      { S7_Templates := "SrcType := DInt" } EQ_Contact(in1 := "Unit1.Em6.ControlNodes".hotPressLeft.sequence.status.currentStep, in2 := #JOB_2_STEP_40)
      Contact( "Unit1.Em6.ControlNodes".hotPressLeft.sequence.status.seqActive )
      wire#w1
      Contact( "Unit1.EmNodes".emRelations.em05.isLinked )
      Coil( "Unit1.Em6.ControlNodes".hotPressLeft."step".action1[240] )
   END_RUNG
   RUNG wire#w1
      Contact( "Unit1.EmNodes".emRelations.em05.sequence.transferPnPLeft.jobInterface.hotPressLeftPLACEJob3_A.unLoadingDone )
      wire#w2
      Contact( true )
      wire#w3
      { S7_Templates := "SrcType := Variant" } NE_Contact(in1 := #NoDataCheck, in2 := "Unit1.EmData".partData[6])
      wire#w4
      Coil( "Unit1.Em6.ControlNodes".hotPressLeft."step".transition1[240] )
   END_RUNG
   RUNG wire#w1
      Contact( "Unit1.Em6.ControlNodes".hotPressLeft."step".transition1[240] )
   END_RUNG wire#w2
   RUNG wire#w1
      I_Contact( "Unit1.EmNodes".emRelations.em05.isLinked )
   END_RUNG wire#w2
   RUNG wire#w3
      I_Contact( "Unit1.Test"."Bool"[40] )
   END_RUNG wire#w4
   RUNG wire#w1
      Contact( "Unit1.Em6.ControlNodes".hotPressLeft."step".transition1[240] )
      { S7_Templates := "time_type := Time" } #statTonTime[240].TON(pt := T#500ms, et =>)
      Move(in := #JOB_2_STEP_50, out1 => "Unit1.Em6.ControlNodes".hotPressLeft.sequence.status.nextStep)
   END_RUNG
   // the same network as SCL:
   #_w1 := ("Unit1.Em6.ControlNodes".hotPressLeft.sequence.status.currentStep = #JOB_2_STEP_40) AND "Unit1.Em6.ControlNodes".hotPressLeft.sequence.status.seqActive;
   "Unit1.Em6.ControlNodes".hotPressLeft."step".action1[240] := #_w1 AND "Unit1.EmNodes".emRelations.em05.isLinked;
   "Unit1.Em6.ControlNodes".hotPressLeft."step".transition1[240] := #_w1 AND ("Unit1.EmNodes".emRelations.em05.sequence.transferPnPLeft.jobInterface.hotPressLeftPLACEJob3_A.unLoadingDone OR "Unit1.Em6.ControlNodes".hotPressLeft."step".transition1[240] OR NOT "Unit1.EmNodes".emRelations.em05.isLinked) AND true AND ((#NoDataCheck <> "Unit1.EmData".partData[6]) OR NOT "Unit1.Test"."Bool"[40]);
   #statTonTime[240].TON(IN := #_w1 AND "Unit1.Em6.ControlNodes".hotPressLeft."step".transition1[240],
                         PT := T#500ms);
   IF #statTonTime[240].Q THEN
       "Unit1.Em6.ControlNodes".hotPressLeft.sequence.status.nextStep := #JOB_2_STEP_50;
   END_IF;
END_REGION

REGION Network 21: Step[250] : Spare
   RUNG wire#powerrail
      { S7_Templates := "SrcType := DInt" } EQ_Contact(in1 := "Unit1.Em6.ControlNodes".hotPressLeft.sequence.status.currentStep, in2 := #JOB_2_STEP_50)
      Contact( "Unit1.Em6.ControlNodes".hotPressLeft.sequence.status.seqActive )
      wire#w1
      Coil( "Unit1.Em6.ControlNodes".hotPressLeft."step".action1[250] )
   END_RUNG
   RUNG wire#w1
      Coil( "Unit1.Em6.ControlNodes".hotPressLeft."step".transition1[250] )
   END_RUNG
   RUNG wire#w1
      Contact( "Unit1.Em6.ControlNodes".hotPressLeft."step".transition1[250] )
      { S7_Templates := "time_type := Time" } #statTonTime[250].TON(pt := T#0ms, et =>)
      Move(in := #JOB_2_STEP_90, out1 => "Unit1.Em6.ControlNodes".hotPressLeft.sequence.status.nextStep)
   END_RUNG
   // the same network as SCL:
   "Unit1.Em6.ControlNodes".hotPressLeft."step".action1[250] := ("Unit1.Em6.ControlNodes".hotPressLeft.sequence.status.currentStep = #JOB_2_STEP_50) AND "Unit1.Em6.ControlNodes".hotPressLeft.sequence.status.seqActive;
   "Unit1.Em6.ControlNodes".hotPressLeft."step".transition1[250] := ("Unit1.Em6.ControlNodes".hotPressLeft.sequence.status.currentStep = #JOB_2_STEP_50) AND "Unit1.Em6.ControlNodes".hotPressLeft.sequence.status.seqActive;
   #statTonTime[250].TON(IN := ("Unit1.Em6.ControlNodes".hotPressLeft.sequence.status.currentStep = #JOB_2_STEP_50) AND "Unit1.Em6.ControlNodes".hotPressLeft.sequence.status.seqActive AND "Unit1.Em6.ControlNodes".hotPressLeft."step".transition1[250],
                         PT := T#0ms);
   IF #statTonTime[250].Q THEN
       "Unit1.Em6.ControlNodes".hotPressLeft.sequence.status.nextStep := #JOB_2_STEP_90;
   END_IF;
END_REGION

REGION Network 22: Step[290] : JOB[2] Step End
   RUNG wire#powerrail
      { S7_Templates := "SrcType := DInt" } EQ_Contact(in1 := "Unit1.Em6.ControlNodes".hotPressLeft.sequence.status.currentStep, in2 := #JOB_2_STEP_90)
      Contact( "Unit1.Em6.ControlNodes".hotPressLeft.sequence.status.seqActive )
      wire#w1
      Coil( "Unit1.Em6.ControlNodes".hotPressLeft."step".action1[290] )
   END_RUNG
   RUNG wire#w1
      Coil( "Unit1.Em6.ControlNodes".hotPressLeft."step".transition1[290] )
   END_RUNG
   RUNG wire#w1
      Contact( "Unit1.Em6.ControlNodes".hotPressLeft."step".transition1[290] )
      { S7_Templates := "time_type := Time" } #statTonTime[290].TON(pt := T#100ms, et =>)
      Move(in := #STEP_IDLE, out1 => "Unit1.Em6.ControlNodes".hotPressLeft.sequence.status.nextStep)
   END_RUNG
   // the same network as SCL:
   "Unit1.Em6.ControlNodes".hotPressLeft."step".action1[290] := ("Unit1.Em6.ControlNodes".hotPressLeft.sequence.status.currentStep = #JOB_2_STEP_90) AND "Unit1.Em6.ControlNodes".hotPressLeft.sequence.status.seqActive;
   "Unit1.Em6.ControlNodes".hotPressLeft."step".transition1[290] := ("Unit1.Em6.ControlNodes".hotPressLeft.sequence.status.currentStep = #JOB_2_STEP_90) AND "Unit1.Em6.ControlNodes".hotPressLeft.sequence.status.seqActive;
   #statTonTime[290].TON(IN := ("Unit1.Em6.ControlNodes".hotPressLeft.sequence.status.currentStep = #JOB_2_STEP_90) AND "Unit1.Em6.ControlNodes".hotPressLeft.sequence.status.seqActive AND "Unit1.Em6.ControlNodes".hotPressLeft."step".transition1[290],
                         PT := T#100ms);
   IF #statTonTime[290].Q THEN
       "Unit1.Em6.ControlNodes".hotPressLeft.sequence.status.nextStep := #STEP_IDLE;
   END_IF;
END_REGION

REGION Network 23: *************** JOB[3] JR HOT PRESS=AUTO *****************
END_REGION

REGION Network 24: Step[301] : JOB[3] Condition
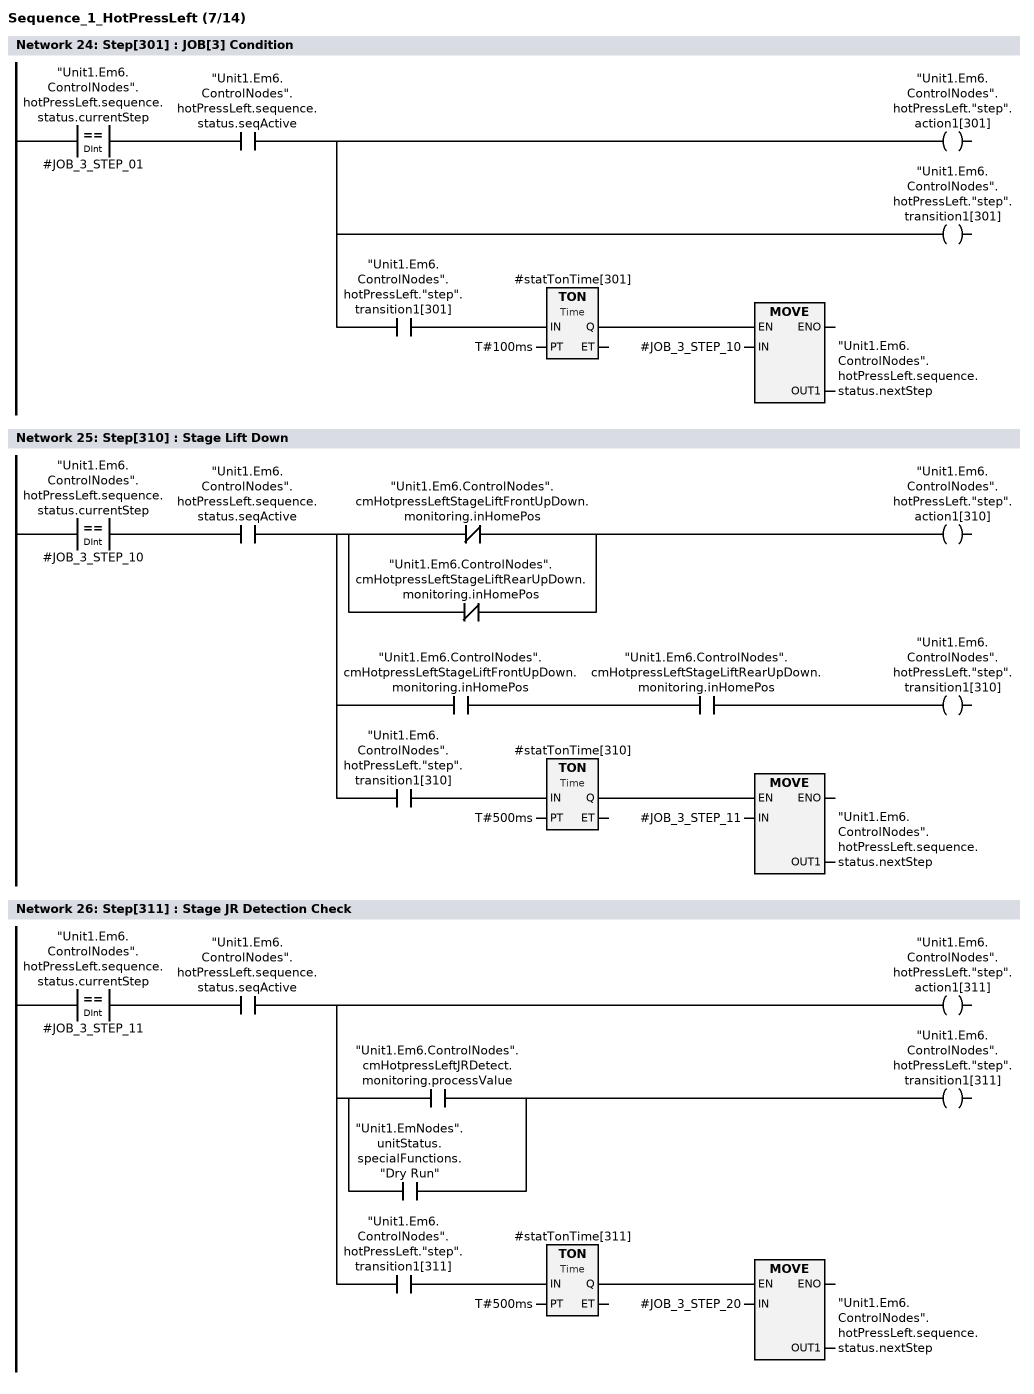
   RUNG wire#powerrail
      { S7_Templates := "SrcType := DInt" } EQ_Contact(in1 := "Unit1.Em6.ControlNodes".hotPressLeft.sequence.status.currentStep, in2 := #JOB_3_STEP_01)
      Contact( "Unit1.Em6.ControlNodes".hotPressLeft.sequence.status.seqActive )
      wire#w1
      Coil( "Unit1.Em6.ControlNodes".hotPressLeft."step".action1[301] )
   END_RUNG
   RUNG wire#w1
      Coil( "Unit1.Em6.ControlNodes".hotPressLeft."step".transition1[301] )
   END_RUNG
   RUNG wire#w1
      Contact( "Unit1.Em6.ControlNodes".hotPressLeft."step".transition1[301] )
      { S7_Templates := "time_type := Time" } #statTonTime[301].TON(pt := T#100ms, et =>)
      Move(in := #JOB_3_STEP_10, out1 => "Unit1.Em6.ControlNodes".hotPressLeft.sequence.status.nextStep)
   END_RUNG
   // the same network as SCL:
   "Unit1.Em6.ControlNodes".hotPressLeft."step".action1[301] := ("Unit1.Em6.ControlNodes".hotPressLeft.sequence.status.currentStep = #JOB_3_STEP_01) AND "Unit1.Em6.ControlNodes".hotPressLeft.sequence.status.seqActive;
   "Unit1.Em6.ControlNodes".hotPressLeft."step".transition1[301] := ("Unit1.Em6.ControlNodes".hotPressLeft.sequence.status.currentStep = #JOB_3_STEP_01) AND "Unit1.Em6.ControlNodes".hotPressLeft.sequence.status.seqActive;
   #statTonTime[301].TON(IN := ("Unit1.Em6.ControlNodes".hotPressLeft.sequence.status.currentStep = #JOB_3_STEP_01) AND "Unit1.Em6.ControlNodes".hotPressLeft.sequence.status.seqActive AND "Unit1.Em6.ControlNodes".hotPressLeft."step".transition1[301],
                         PT := T#100ms);
   IF #statTonTime[301].Q THEN
       "Unit1.Em6.ControlNodes".hotPressLeft.sequence.status.nextStep := #JOB_3_STEP_10;
   END_IF;
END_REGION

REGION Network 25: Step[310] : Stage Lift Down
   RUNG wire#powerrail
      { S7_Templates := "SrcType := DInt" } EQ_Contact(in1 := "Unit1.Em6.ControlNodes".hotPressLeft.sequence.status.currentStep, in2 := #JOB_3_STEP_10)
      Contact( "Unit1.Em6.ControlNodes".hotPressLeft.sequence.status.seqActive )
      wire#w1
      I_Contact( "Unit1.Em6.ControlNodes".cmHotpressLeftStageLiftFrontUpDown.monitoring.inHomePos )
      wire#w2
      Coil( "Unit1.Em6.ControlNodes".hotPressLeft."step".action1[310] )
   END_RUNG
   RUNG wire#w1
      I_Contact( "Unit1.Em6.ControlNodes".cmHotpressLeftStageLiftRearUpDown.monitoring.inHomePos )
   END_RUNG wire#w2
   RUNG wire#w1
      Contact( "Unit1.Em6.ControlNodes".cmHotpressLeftStageLiftFrontUpDown.monitoring.inHomePos )
      Contact( "Unit1.Em6.ControlNodes".cmHotpressLeftStageLiftRearUpDown.monitoring.inHomePos )
      Coil( "Unit1.Em6.ControlNodes".hotPressLeft."step".transition1[310] )
   END_RUNG
   RUNG wire#w1
      Contact( "Unit1.Em6.ControlNodes".hotPressLeft."step".transition1[310] )
      { S7_Templates := "time_type := Time" } #statTonTime[310].TON(pt := T#500ms, et =>)
      Move(in := #JOB_3_STEP_11, out1 => "Unit1.Em6.ControlNodes".hotPressLeft.sequence.status.nextStep)
   END_RUNG
   // the same network as SCL:
   #_w1 := ("Unit1.Em6.ControlNodes".hotPressLeft.sequence.status.currentStep = #JOB_3_STEP_10) AND "Unit1.Em6.ControlNodes".hotPressLeft.sequence.status.seqActive;
   "Unit1.Em6.ControlNodes".hotPressLeft."step".action1[310] := #_w1 AND (NOT "Unit1.Em6.ControlNodes".cmHotpressLeftStageLiftFrontUpDown.monitoring.inHomePos OR NOT "Unit1.Em6.ControlNodes".cmHotpressLeftStageLiftRearUpDown.monitoring.inHomePos);
   "Unit1.Em6.ControlNodes".hotPressLeft."step".transition1[310] := #_w1 AND "Unit1.Em6.ControlNodes".cmHotpressLeftStageLiftFrontUpDown.monitoring.inHomePos AND "Unit1.Em6.ControlNodes".cmHotpressLeftStageLiftRearUpDown.monitoring.inHomePos;
   #statTonTime[310].TON(IN := #_w1 AND "Unit1.Em6.ControlNodes".hotPressLeft."step".transition1[310],
                         PT := T#500ms);
   IF #statTonTime[310].Q THEN
       "Unit1.Em6.ControlNodes".hotPressLeft.sequence.status.nextStep := #JOB_3_STEP_11;
   END_IF;
END_REGION

REGION Network 26: Step[311] : Stage JR Detection Check
   RUNG wire#powerrail
      { S7_Templates := "SrcType := DInt" } EQ_Contact(in1 := "Unit1.Em6.ControlNodes".hotPressLeft.sequence.status.currentStep, in2 := #JOB_3_STEP_11)
      Contact( "Unit1.Em6.ControlNodes".hotPressLeft.sequence.status.seqActive )
      wire#w1
      Coil( "Unit1.Em6.ControlNodes".hotPressLeft."step".action1[311] )
   END_RUNG
   RUNG wire#w1
      Contact( "Unit1.Em6.ControlNodes".cmHotpressLeftJRDetect.monitoring.processValue )
      wire#w2
      Coil( "Unit1.Em6.ControlNodes".hotPressLeft."step".transition1[311] )
   END_RUNG
   RUNG wire#w1
      Contact( "Unit1.EmNodes".unitStatus.specialFunctions."Dry Run" )
   END_RUNG wire#w2
   RUNG wire#w1
      Contact( "Unit1.Em6.ControlNodes".hotPressLeft."step".transition1[311] )
      { S7_Templates := "time_type := Time" } #statTonTime[311].TON(pt := T#500ms, et =>)
      Move(in := #JOB_3_STEP_20, out1 => "Unit1.Em6.ControlNodes".hotPressLeft.sequence.status.nextStep)
   END_RUNG
   // the same network as SCL:
   "Unit1.Em6.ControlNodes".hotPressLeft."step".action1[311] := ("Unit1.Em6.ControlNodes".hotPressLeft.sequence.status.currentStep = #JOB_3_STEP_11) AND "Unit1.Em6.ControlNodes".hotPressLeft.sequence.status.seqActive;
   "Unit1.Em6.ControlNodes".hotPressLeft."step".transition1[311] := ("Unit1.Em6.ControlNodes".hotPressLeft.sequence.status.currentStep = #JOB_3_STEP_11) AND "Unit1.Em6.ControlNodes".hotPressLeft.sequence.status.seqActive AND ("Unit1.Em6.ControlNodes".cmHotpressLeftJRDetect.monitoring.processValue OR "Unit1.EmNodes".unitStatus.specialFunctions."Dry Run");
   #statTonTime[311].TON(IN := ("Unit1.Em6.ControlNodes".hotPressLeft.sequence.status.currentStep = #JOB_3_STEP_11) AND "Unit1.Em6.ControlNodes".hotPressLeft.sequence.status.seqActive AND "Unit1.Em6.ControlNodes".hotPressLeft."step".transition1[311],
                         PT := T#500ms);
   IF #statTonTime[311].Q THEN
       "Unit1.Em6.ControlNodes".hotPressLeft.sequence.status.nextStep := #JOB_3_STEP_20;
   END_IF;
END_REGION

REGION Network 27: Step[320] : Spare
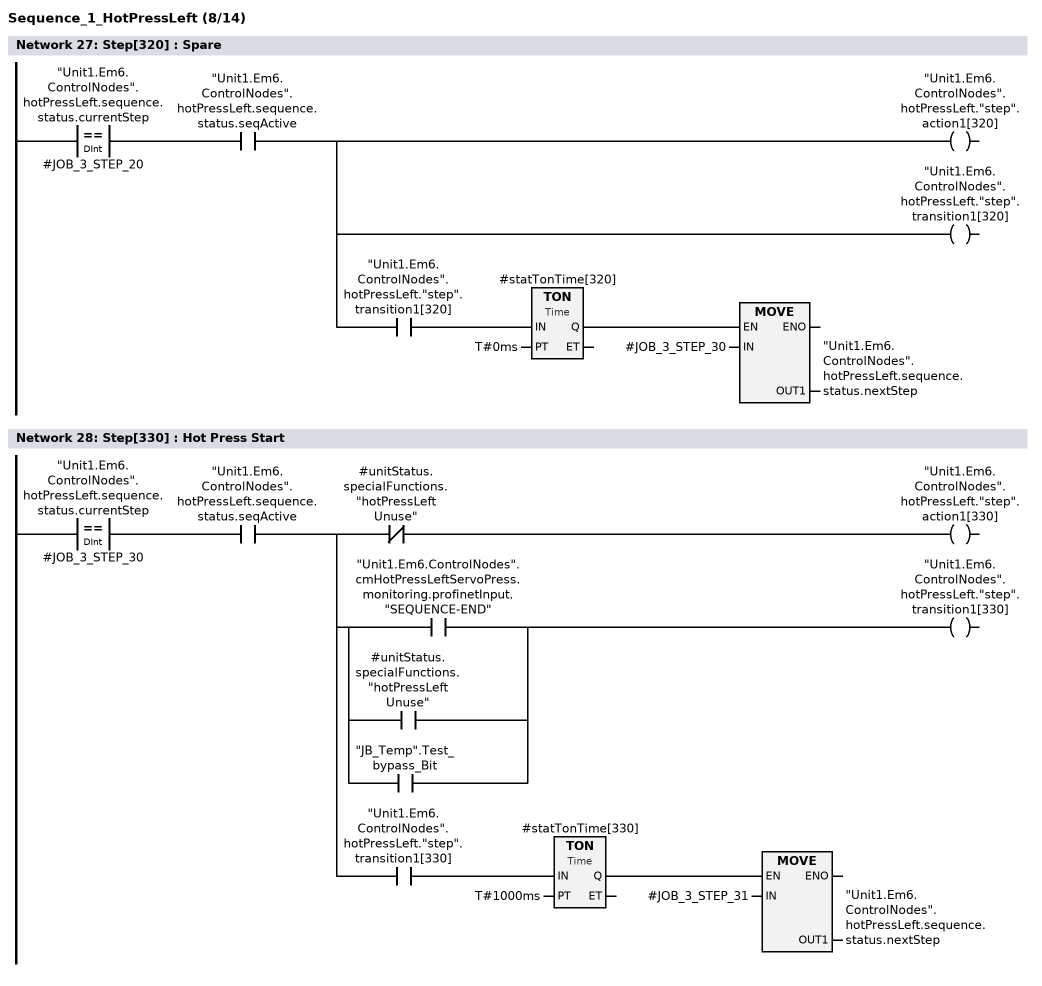
   RUNG wire#powerrail
      { S7_Templates := "SrcType := DInt" } EQ_Contact(in1 := "Unit1.Em6.ControlNodes".hotPressLeft.sequence.status.currentStep, in2 := #JOB_3_STEP_20)
      Contact( "Unit1.Em6.ControlNodes".hotPressLeft.sequence.status.seqActive )
      wire#w1
      Coil( "Unit1.Em6.ControlNodes".hotPressLeft."step".action1[320] )
   END_RUNG
   RUNG wire#w1
      Coil( "Unit1.Em6.ControlNodes".hotPressLeft."step".transition1[320] )
   END_RUNG
   RUNG wire#w1
      Contact( "Unit1.Em6.ControlNodes".hotPressLeft."step".transition1[320] )
      { S7_Templates := "time_type := Time" } #statTonTime[320].TON(pt := T#0ms, et =>)
      Move(in := #JOB_3_STEP_30, out1 => "Unit1.Em6.ControlNodes".hotPressLeft.sequence.status.nextStep)
   END_RUNG
   // the same network as SCL:
   "Unit1.Em6.ControlNodes".hotPressLeft."step".action1[320] := ("Unit1.Em6.ControlNodes".hotPressLeft.sequence.status.currentStep = #JOB_3_STEP_20) AND "Unit1.Em6.ControlNodes".hotPressLeft.sequence.status.seqActive;
   "Unit1.Em6.ControlNodes".hotPressLeft."step".transition1[320] := ("Unit1.Em6.ControlNodes".hotPressLeft.sequence.status.currentStep = #JOB_3_STEP_20) AND "Unit1.Em6.ControlNodes".hotPressLeft.sequence.status.seqActive;
   #statTonTime[320].TON(IN := ("Unit1.Em6.ControlNodes".hotPressLeft.sequence.status.currentStep = #JOB_3_STEP_20) AND "Unit1.Em6.ControlNodes".hotPressLeft.sequence.status.seqActive AND "Unit1.Em6.ControlNodes".hotPressLeft."step".transition1[320],
                         PT := T#0ms);
   IF #statTonTime[320].Q THEN
       "Unit1.Em6.ControlNodes".hotPressLeft.sequence.status.nextStep := #JOB_3_STEP_30;
   END_IF;
END_REGION

REGION Network 28: Step[330] : Hot Press Start
   RUNG wire#powerrail
      { S7_Templates := "SrcType := DInt" } EQ_Contact(in1 := "Unit1.Em6.ControlNodes".hotPressLeft.sequence.status.currentStep, in2 := #JOB_3_STEP_30)
      Contact( "Unit1.Em6.ControlNodes".hotPressLeft.sequence.status.seqActive )
      wire#w1
      I_Contact( #unitStatus.specialFunctions."hotPressLeft Unuse" )
      Coil( "Unit1.Em6.ControlNodes".hotPressLeft."step".action1[330] )
   END_RUNG
   RUNG wire#w1
      Contact( "Unit1.Em6.ControlNodes".cmHotPressLeftServoPress.monitoring.profinetInput."SEQUENCE-END" )
      wire#w2
      Coil( "Unit1.Em6.ControlNodes".hotPressLeft."step".transition1[330] )
   END_RUNG
   RUNG wire#w1
      Contact( #unitStatus.specialFunctions."hotPressLeft Unuse" )
   END_RUNG wire#w2
   RUNG wire#w1
      Contact( "JB_Temp".Test_bypass_Bit )
   END_RUNG wire#w2
   RUNG wire#w1
      Contact( "Unit1.Em6.ControlNodes".hotPressLeft."step".transition1[330] )
      { S7_Templates := "time_type := Time" } #statTonTime[330].TON(pt := T#1000ms, et =>)
      Move(in := #JOB_3_STEP_31, out1 => "Unit1.Em6.ControlNodes".hotPressLeft.sequence.status.nextStep)
   END_RUNG
   // the same network as SCL:
   #_w1 := ("Unit1.Em6.ControlNodes".hotPressLeft.sequence.status.currentStep = #JOB_3_STEP_30) AND "Unit1.Em6.ControlNodes".hotPressLeft.sequence.status.seqActive;
   "Unit1.Em6.ControlNodes".hotPressLeft."step".action1[330] := #_w1 AND NOT #unitStatus.specialFunctions."hotPressLeft Unuse";
   "Unit1.Em6.ControlNodes".hotPressLeft."step".transition1[330] := #_w1 AND ("Unit1.Em6.ControlNodes".cmHotPressLeftServoPress.monitoring.profinetInput."SEQUENCE-END" OR #unitStatus.specialFunctions."hotPressLeft Unuse" OR "JB_Temp".Test_bypass_Bit);
   #statTonTime[330].TON(IN := #_w1 AND "Unit1.Em6.ControlNodes".hotPressLeft."step".transition1[330],
                         PT := T#1000ms);
   IF #statTonTime[330].Q THEN
       "Unit1.Em6.ControlNodes".hotPressLeft.sequence.status.nextStep := #JOB_3_STEP_31;
   END_IF;
END_REGION

REGION Network 29: Step[331] : Hot Press Result
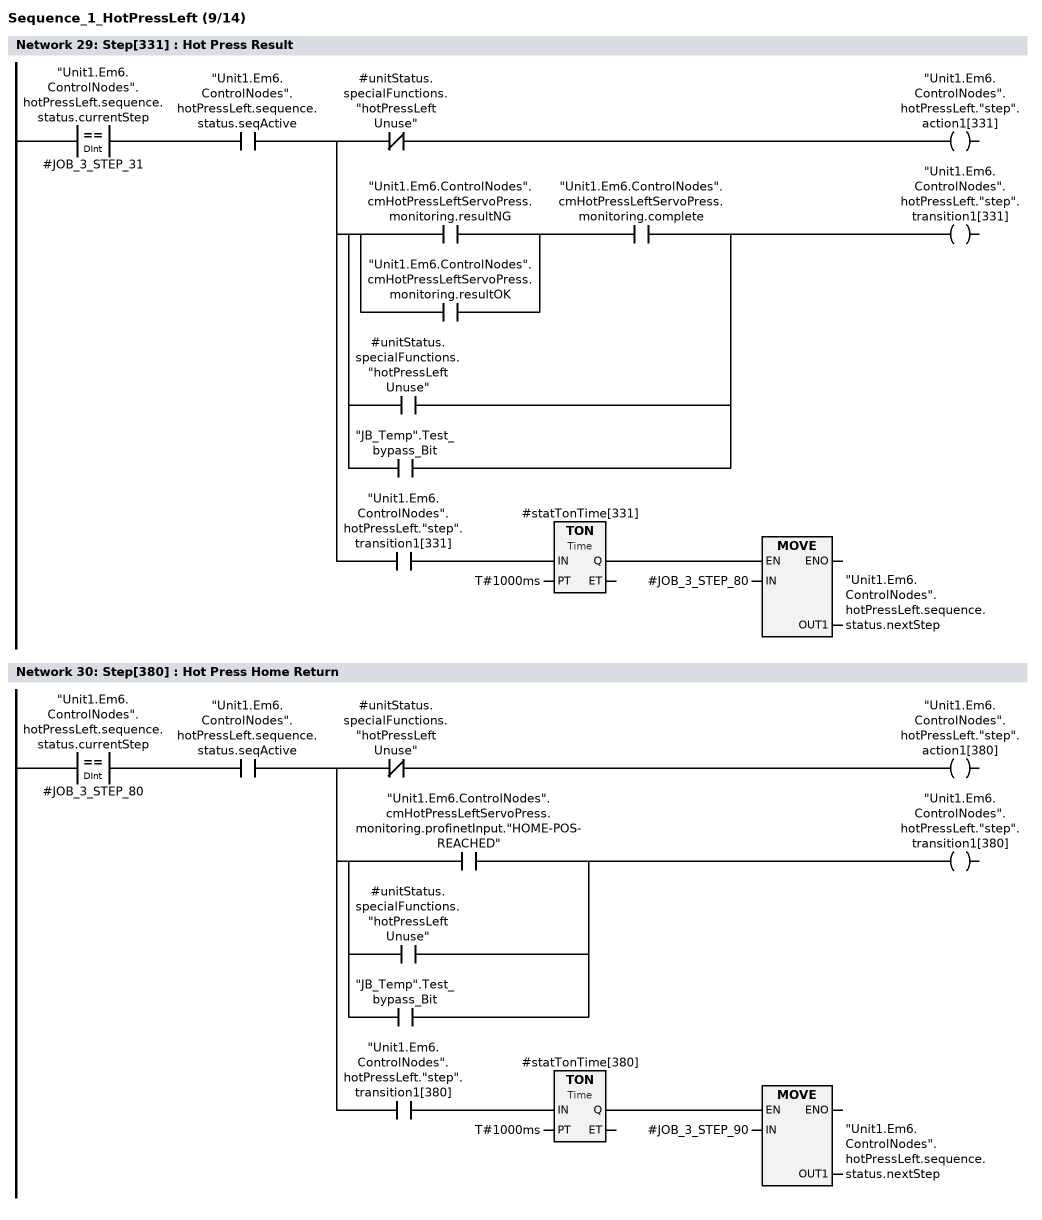
   RUNG wire#powerrail
      { S7_Templates := "SrcType := DInt" } EQ_Contact(in1 := "Unit1.Em6.ControlNodes".hotPressLeft.sequence.status.currentStep, in2 := #JOB_3_STEP_31)
      Contact( "Unit1.Em6.ControlNodes".hotPressLeft.sequence.status.seqActive )
      wire#w1
      I_Contact( #unitStatus.specialFunctions."hotPressLeft Unuse" )
      Coil( "Unit1.Em6.ControlNodes".hotPressLeft."step".action1[331] )
   END_RUNG
   RUNG wire#w1
      Contact( "Unit1.Em6.ControlNodes".cmHotPressLeftServoPress.monitoring.resultNG )
      wire#w2
      Contact( "Unit1.Em6.ControlNodes".cmHotPressLeftServoPress.monitoring.complete )
      wire#w3
      Coil( "Unit1.Em6.ControlNodes".hotPressLeft."step".transition1[331] )
   END_RUNG
   RUNG wire#w1
      Contact( "Unit1.Em6.ControlNodes".cmHotPressLeftServoPress.monitoring.resultOK )
   END_RUNG wire#w2
   RUNG wire#w1
      Contact( #unitStatus.specialFunctions."hotPressLeft Unuse" )
   END_RUNG wire#w3
   RUNG wire#w1
      Contact( "JB_Temp".Test_bypass_Bit )
   END_RUNG wire#w3
   RUNG wire#w1
      Contact( "Unit1.Em6.ControlNodes".hotPressLeft."step".transition1[331] )
      { S7_Templates := "time_type := Time" } #statTonTime[331].TON(pt := T#1000ms, et =>)
      Move(in := #JOB_3_STEP_80, out1 => "Unit1.Em6.ControlNodes".hotPressLeft.sequence.status.nextStep)
   END_RUNG
   // the same network as SCL:
   #_w1 := ("Unit1.Em6.ControlNodes".hotPressLeft.sequence.status.currentStep = #JOB_3_STEP_31) AND "Unit1.Em6.ControlNodes".hotPressLeft.sequence.status.seqActive;
   "Unit1.Em6.ControlNodes".hotPressLeft."step".action1[331] := #_w1 AND NOT #unitStatus.specialFunctions."hotPressLeft Unuse";
   "Unit1.Em6.ControlNodes".hotPressLeft."step".transition1[331] := #_w1 AND ((("Unit1.Em6.ControlNodes".cmHotPressLeftServoPress.monitoring.resultNG OR "Unit1.Em6.ControlNodes".cmHotPressLeftServoPress.monitoring.resultOK) AND "Unit1.Em6.ControlNodes".cmHotPressLeftServoPress.monitoring.complete) OR #unitStatus.specialFunctions."hotPressLeft Unuse" OR "JB_Temp".Test_bypass_Bit);
   #statTonTime[331].TON(IN := #_w1 AND "Unit1.Em6.ControlNodes".hotPressLeft."step".transition1[331],
                         PT := T#1000ms);
   IF #statTonTime[331].Q THEN
       "Unit1.Em6.ControlNodes".hotPressLeft.sequence.status.nextStep := #JOB_3_STEP_80;
   END_IF;
END_REGION

REGION Network 30: Step[380] : Hot Press Home Return
   RUNG wire#powerrail
      { S7_Templates := "SrcType := DInt" } EQ_Contact(in1 := "Unit1.Em6.ControlNodes".hotPressLeft.sequence.status.currentStep, in2 := #JOB_3_STEP_80)
      Contact( "Unit1.Em6.ControlNodes".hotPressLeft.sequence.status.seqActive )
      wire#w1
      I_Contact( #unitStatus.specialFunctions."hotPressLeft Unuse" )
      Coil( "Unit1.Em6.ControlNodes".hotPressLeft."step".action1[380] )
   END_RUNG
   RUNG wire#w1
      Contact( "Unit1.Em6.ControlNodes".cmHotPressLeftServoPress.monitoring.profinetInput."HOME-POS-REACHED" )
      wire#w2
      Coil( "Unit1.Em6.ControlNodes".hotPressLeft."step".transition1[380] )
   END_RUNG
   RUNG wire#w1
      Contact( #unitStatus.specialFunctions."hotPressLeft Unuse" )
   END_RUNG wire#w2
   RUNG wire#w1
      Contact( "JB_Temp".Test_bypass_Bit )
   END_RUNG wire#w2
   RUNG wire#w1
      Contact( "Unit1.Em6.ControlNodes".hotPressLeft."step".transition1[380] )
      { S7_Templates := "time_type := Time" } #statTonTime[380].TON(pt := T#1000ms, et =>)
      Move(in := #JOB_3_STEP_90, out1 => "Unit1.Em6.ControlNodes".hotPressLeft.sequence.status.nextStep)
   END_RUNG
   // the same network as SCL:
   #_w1 := ("Unit1.Em6.ControlNodes".hotPressLeft.sequence.status.currentStep = #JOB_3_STEP_80) AND "Unit1.Em6.ControlNodes".hotPressLeft.sequence.status.seqActive;
   "Unit1.Em6.ControlNodes".hotPressLeft."step".action1[380] := #_w1 AND NOT #unitStatus.specialFunctions."hotPressLeft Unuse";
   "Unit1.Em6.ControlNodes".hotPressLeft."step".transition1[380] := #_w1 AND ("Unit1.Em6.ControlNodes".cmHotPressLeftServoPress.monitoring.profinetInput."HOME-POS-REACHED" OR #unitStatus.specialFunctions."hotPressLeft Unuse" OR "JB_Temp".Test_bypass_Bit);
   #statTonTime[380].TON(IN := #_w1 AND "Unit1.Em6.ControlNodes".hotPressLeft."step".transition1[380],
                         PT := T#1000ms);
   IF #statTonTime[380].Q THEN
       "Unit1.Em6.ControlNodes".hotPressLeft.sequence.status.nextStep := #JOB_3_STEP_90;
   END_IF;
END_REGION

REGION Network 31: Step[390] : JOB[3] Step End
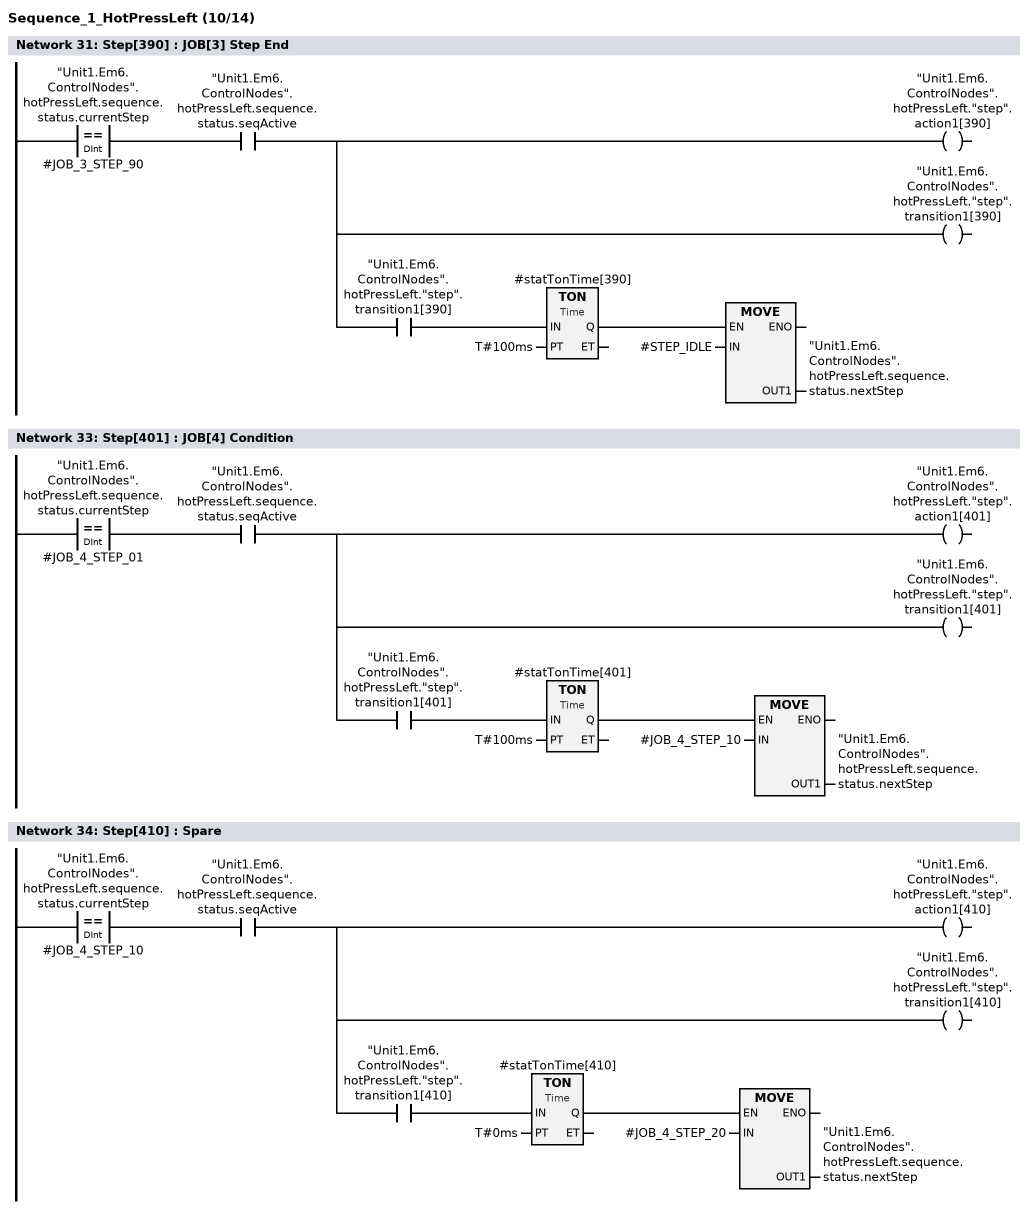
   RUNG wire#powerrail
      { S7_Templates := "SrcType := DInt" } EQ_Contact(in1 := "Unit1.Em6.ControlNodes".hotPressLeft.sequence.status.currentStep, in2 := #JOB_3_STEP_90)
      Contact( "Unit1.Em6.ControlNodes".hotPressLeft.sequence.status.seqActive )
      wire#w1
      Coil( "Unit1.Em6.ControlNodes".hotPressLeft."step".action1[390] )
   END_RUNG
   RUNG wire#w1
      Coil( "Unit1.Em6.ControlNodes".hotPressLeft."step".transition1[390] )
   END_RUNG
   RUNG wire#w1
      Contact( "Unit1.Em6.ControlNodes".hotPressLeft."step".transition1[390] )
      { S7_Templates := "time_type := Time" } #statTonTime[390].TON(pt := T#100ms, et =>)
      Move(in := #STEP_IDLE, out1 => "Unit1.Em6.ControlNodes".hotPressLeft.sequence.status.nextStep)
   END_RUNG
   // the same network as SCL:
   "Unit1.Em6.ControlNodes".hotPressLeft."step".action1[390] := ("Unit1.Em6.ControlNodes".hotPressLeft.sequence.status.currentStep = #JOB_3_STEP_90) AND "Unit1.Em6.ControlNodes".hotPressLeft.sequence.status.seqActive;
   "Unit1.Em6.ControlNodes".hotPressLeft."step".transition1[390] := ("Unit1.Em6.ControlNodes".hotPressLeft.sequence.status.currentStep = #JOB_3_STEP_90) AND "Unit1.Em6.ControlNodes".hotPressLeft.sequence.status.seqActive;
   #statTonTime[390].TON(IN := ("Unit1.Em6.ControlNodes".hotPressLeft.sequence.status.currentStep = #JOB_3_STEP_90) AND "Unit1.Em6.ControlNodes".hotPressLeft.sequence.status.seqActive AND "Unit1.Em6.ControlNodes".hotPressLeft."step".transition1[390],
                         PT := T#100ms);
   IF #statTonTime[390].Q THEN
       "Unit1.Em6.ControlNodes".hotPressLeft.sequence.status.nextStep := #STEP_IDLE;
   END_IF;
END_REGION

REGION Network 32: *************** JOB[4] JR PUT=AUTO ***********************
END_REGION

REGION Network 33: Step[401] : JOB[4] Condition
   RUNG wire#powerrail
      { S7_Templates := "SrcType := DInt" } EQ_Contact(in1 := "Unit1.Em6.ControlNodes".hotPressLeft.sequence.status.currentStep, in2 := #JOB_4_STEP_01)
      Contact( "Unit1.Em6.ControlNodes".hotPressLeft.sequence.status.seqActive )
      wire#w1
      Coil( "Unit1.Em6.ControlNodes".hotPressLeft."step".action1[401] )
   END_RUNG
   RUNG wire#w1
      Coil( "Unit1.Em6.ControlNodes".hotPressLeft."step".transition1[401] )
   END_RUNG
   RUNG wire#w1
      Contact( "Unit1.Em6.ControlNodes".hotPressLeft."step".transition1[401] )
      { S7_Templates := "time_type := Time" } #statTonTime[401].TON(pt := T#100ms, et =>)
      Move(in := #JOB_4_STEP_10, out1 => "Unit1.Em6.ControlNodes".hotPressLeft.sequence.status.nextStep)
   END_RUNG
   // the same network as SCL:
   "Unit1.Em6.ControlNodes".hotPressLeft."step".action1[401] := ("Unit1.Em6.ControlNodes".hotPressLeft.sequence.status.currentStep = #JOB_4_STEP_01) AND "Unit1.Em6.ControlNodes".hotPressLeft.sequence.status.seqActive;
   "Unit1.Em6.ControlNodes".hotPressLeft."step".transition1[401] := ("Unit1.Em6.ControlNodes".hotPressLeft.sequence.status.currentStep = #JOB_4_STEP_01) AND "Unit1.Em6.ControlNodes".hotPressLeft.sequence.status.seqActive;
   #statTonTime[401].TON(IN := ("Unit1.Em6.ControlNodes".hotPressLeft.sequence.status.currentStep = #JOB_4_STEP_01) AND "Unit1.Em6.ControlNodes".hotPressLeft.sequence.status.seqActive AND "Unit1.Em6.ControlNodes".hotPressLeft."step".transition1[401],
                         PT := T#100ms);
   IF #statTonTime[401].Q THEN
       "Unit1.Em6.ControlNodes".hotPressLeft.sequence.status.nextStep := #JOB_4_STEP_10;
   END_IF;
END_REGION

REGION Network 34: Step[410] : Spare
   RUNG wire#powerrail
      { S7_Templates := "SrcType := DInt" } EQ_Contact(in1 := "Unit1.Em6.ControlNodes".hotPressLeft.sequence.status.currentStep, in2 := #JOB_4_STEP_10)
      Contact( "Unit1.Em6.ControlNodes".hotPressLeft.sequence.status.seqActive )
      wire#w1
      Coil( "Unit1.Em6.ControlNodes".hotPressLeft."step".action1[410] )
   END_RUNG
   RUNG wire#w1
      Coil( "Unit1.Em6.ControlNodes".hotPressLeft."step".transition1[410] )
   END_RUNG
   RUNG wire#w1
      Contact( "Unit1.Em6.ControlNodes".hotPressLeft."step".transition1[410] )
      { S7_Templates := "time_type := Time" } #statTonTime[410].TON(pt := T#0ms, et =>)
      Move(in := #JOB_4_STEP_20, out1 => "Unit1.Em6.ControlNodes".hotPressLeft.sequence.status.nextStep)
   END_RUNG
   // the same network as SCL:
   "Unit1.Em6.ControlNodes".hotPressLeft."step".action1[410] := ("Unit1.Em6.ControlNodes".hotPressLeft.sequence.status.currentStep = #JOB_4_STEP_10) AND "Unit1.Em6.ControlNodes".hotPressLeft.sequence.status.seqActive;
   "Unit1.Em6.ControlNodes".hotPressLeft."step".transition1[410] := ("Unit1.Em6.ControlNodes".hotPressLeft.sequence.status.currentStep = #JOB_4_STEP_10) AND "Unit1.Em6.ControlNodes".hotPressLeft.sequence.status.seqActive;
   #statTonTime[410].TON(IN := ("Unit1.Em6.ControlNodes".hotPressLeft.sequence.status.currentStep = #JOB_4_STEP_10) AND "Unit1.Em6.ControlNodes".hotPressLeft.sequence.status.seqActive AND "Unit1.Em6.ControlNodes".hotPressLeft."step".transition1[410],
                         PT := T#0ms);
   IF #statTonTime[410].Q THEN
       "Unit1.Em6.ControlNodes".hotPressLeft.sequence.status.nextStep := #JOB_4_STEP_20;
   END_IF;
END_REGION

REGION Network 35: Step[420] : Stage Lift Up
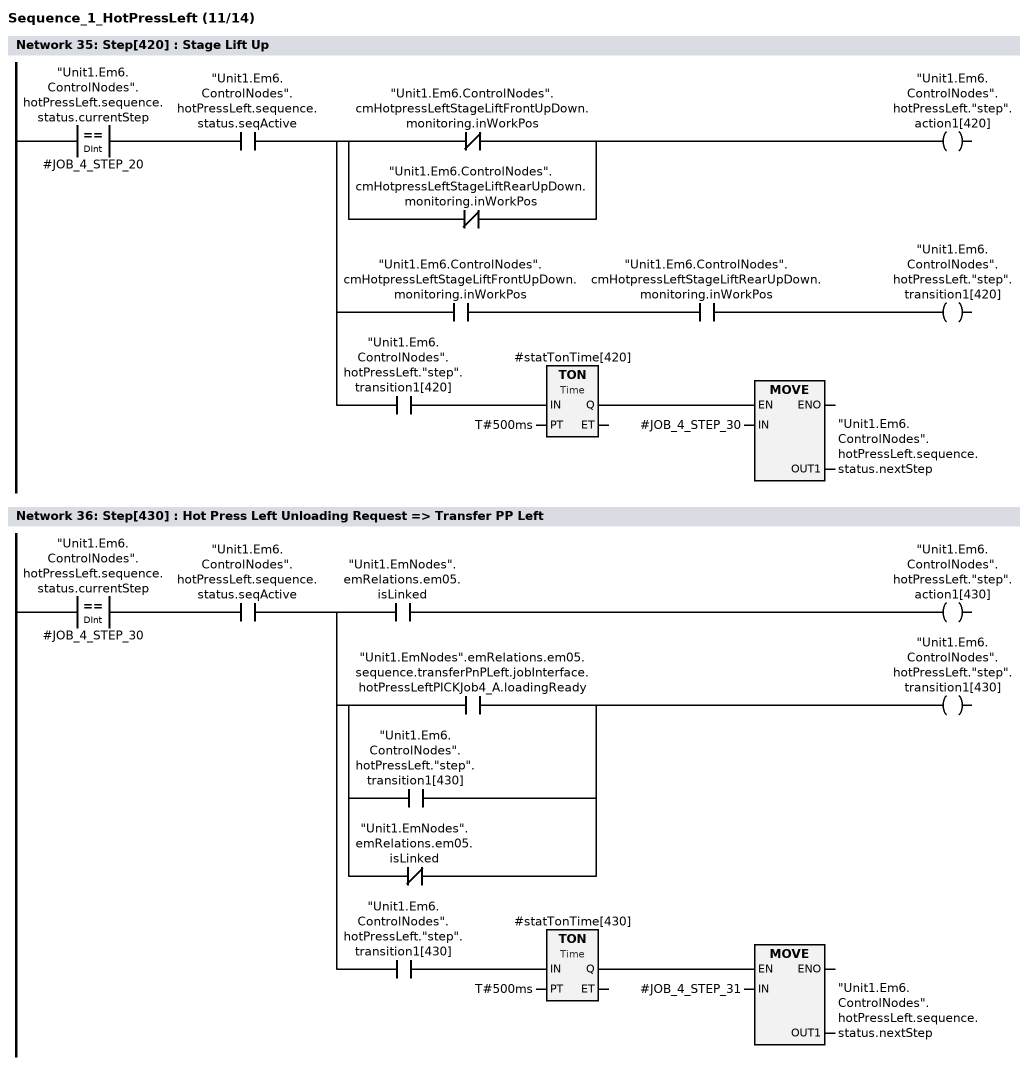
   RUNG wire#powerrail
      { S7_Templates := "SrcType := DInt" } EQ_Contact(in1 := "Unit1.Em6.ControlNodes".hotPressLeft.sequence.status.currentStep, in2 := #JOB_4_STEP_20)
      Contact( "Unit1.Em6.ControlNodes".hotPressLeft.sequence.status.seqActive )
      wire#w1
      I_Contact( "Unit1.Em6.ControlNodes".cmHotpressLeftStageLiftFrontUpDown.monitoring.inWorkPos )
      wire#w2
      Coil( "Unit1.Em6.ControlNodes".hotPressLeft."step".action1[420] )
   END_RUNG
   RUNG wire#w1
      I_Contact( "Unit1.Em6.ControlNodes".cmHotpressLeftStageLiftRearUpDown.monitoring.inWorkPos )
   END_RUNG wire#w2
   RUNG wire#w1
      Contact( "Unit1.Em6.ControlNodes".cmHotpressLeftStageLiftFrontUpDown.monitoring.inWorkPos )
      Contact( "Unit1.Em6.ControlNodes".cmHotpressLeftStageLiftRearUpDown.monitoring.inWorkPos )
      Coil( "Unit1.Em6.ControlNodes".hotPressLeft."step".transition1[420] )
   END_RUNG
   RUNG wire#w1
      Contact( "Unit1.Em6.ControlNodes".hotPressLeft."step".transition1[420] )
      { S7_Templates := "time_type := Time" } #statTonTime[420].TON(pt := T#500ms, et =>)
      Move(in := #JOB_4_STEP_30, out1 => "Unit1.Em6.ControlNodes".hotPressLeft.sequence.status.nextStep)
   END_RUNG
   // the same network as SCL:
   #_w1 := ("Unit1.Em6.ControlNodes".hotPressLeft.sequence.status.currentStep = #JOB_4_STEP_20) AND "Unit1.Em6.ControlNodes".hotPressLeft.sequence.status.seqActive;
   "Unit1.Em6.ControlNodes".hotPressLeft."step".action1[420] := #_w1 AND (NOT "Unit1.Em6.ControlNodes".cmHotpressLeftStageLiftFrontUpDown.monitoring.inWorkPos OR NOT "Unit1.Em6.ControlNodes".cmHotpressLeftStageLiftRearUpDown.monitoring.inWorkPos);
   "Unit1.Em6.ControlNodes".hotPressLeft."step".transition1[420] := #_w1 AND "Unit1.Em6.ControlNodes".cmHotpressLeftStageLiftFrontUpDown.monitoring.inWorkPos AND "Unit1.Em6.ControlNodes".cmHotpressLeftStageLiftRearUpDown.monitoring.inWorkPos;
   #statTonTime[420].TON(IN := #_w1 AND "Unit1.Em6.ControlNodes".hotPressLeft."step".transition1[420],
                         PT := T#500ms);
   IF #statTonTime[420].Q THEN
       "Unit1.Em6.ControlNodes".hotPressLeft.sequence.status.nextStep := #JOB_4_STEP_30;
   END_IF;
END_REGION

REGION Network 36: Step[430] : Hot Press Left Unloading Request => Transfer PP Left
   RUNG wire#powerrail
      { S7_Templates := "SrcType := DInt" } EQ_Contact(in1 := "Unit1.Em6.ControlNodes".hotPressLeft.sequence.status.currentStep, in2 := #JOB_4_STEP_30)
      Contact( "Unit1.Em6.ControlNodes".hotPressLeft.sequence.status.seqActive )
      wire#w1
      Contact( "Unit1.EmNodes".emRelations.em05.isLinked )
      Coil( "Unit1.Em6.ControlNodes".hotPressLeft."step".action1[430] )
   END_RUNG
   RUNG wire#w1
      Contact( "Unit1.EmNodes".emRelations.em05.sequence.transferPnPLeft.jobInterface.hotPressLeftPICKJob4_A.loadingReady )
      wire#w2
      Coil( "Unit1.Em6.ControlNodes".hotPressLeft."step".transition1[430] )
   END_RUNG
   RUNG wire#w1
      Contact( "Unit1.Em6.ControlNodes".hotPressLeft."step".transition1[430] )
   END_RUNG wire#w2
   RUNG wire#w1
      I_Contact( "Unit1.EmNodes".emRelations.em05.isLinked )
   END_RUNG wire#w2
   RUNG wire#w1
      Contact( "Unit1.Em6.ControlNodes".hotPressLeft."step".transition1[430] )
      { S7_Templates := "time_type := Time" } #statTonTime[430].TON(pt := T#500ms, et =>)
      Move(in := #JOB_4_STEP_31, out1 => "Unit1.Em6.ControlNodes".hotPressLeft.sequence.status.nextStep)
   END_RUNG
   // the same network as SCL:
   #_w1 := ("Unit1.Em6.ControlNodes".hotPressLeft.sequence.status.currentStep = #JOB_4_STEP_30) AND "Unit1.Em6.ControlNodes".hotPressLeft.sequence.status.seqActive;
   "Unit1.Em6.ControlNodes".hotPressLeft."step".action1[430] := #_w1 AND "Unit1.EmNodes".emRelations.em05.isLinked;
   "Unit1.Em6.ControlNodes".hotPressLeft."step".transition1[430] := #_w1 AND ("Unit1.EmNodes".emRelations.em05.sequence.transferPnPLeft.jobInterface.hotPressLeftPICKJob4_A.loadingReady OR "Unit1.Em6.ControlNodes".hotPressLeft."step".transition1[430] OR NOT "Unit1.EmNodes".emRelations.em05.isLinked);
   #statTonTime[430].TON(IN := #_w1 AND "Unit1.Em6.ControlNodes".hotPressLeft."step".transition1[430],
                         PT := T#500ms);
   IF #statTonTime[430].Q THEN
       "Unit1.Em6.ControlNodes".hotPressLeft.sequence.status.nextStep := #JOB_4_STEP_31;
   END_IF;
END_REGION

REGION Network 37: Step[431] : Hot Press Left Unloading Check => Transfer PP Left
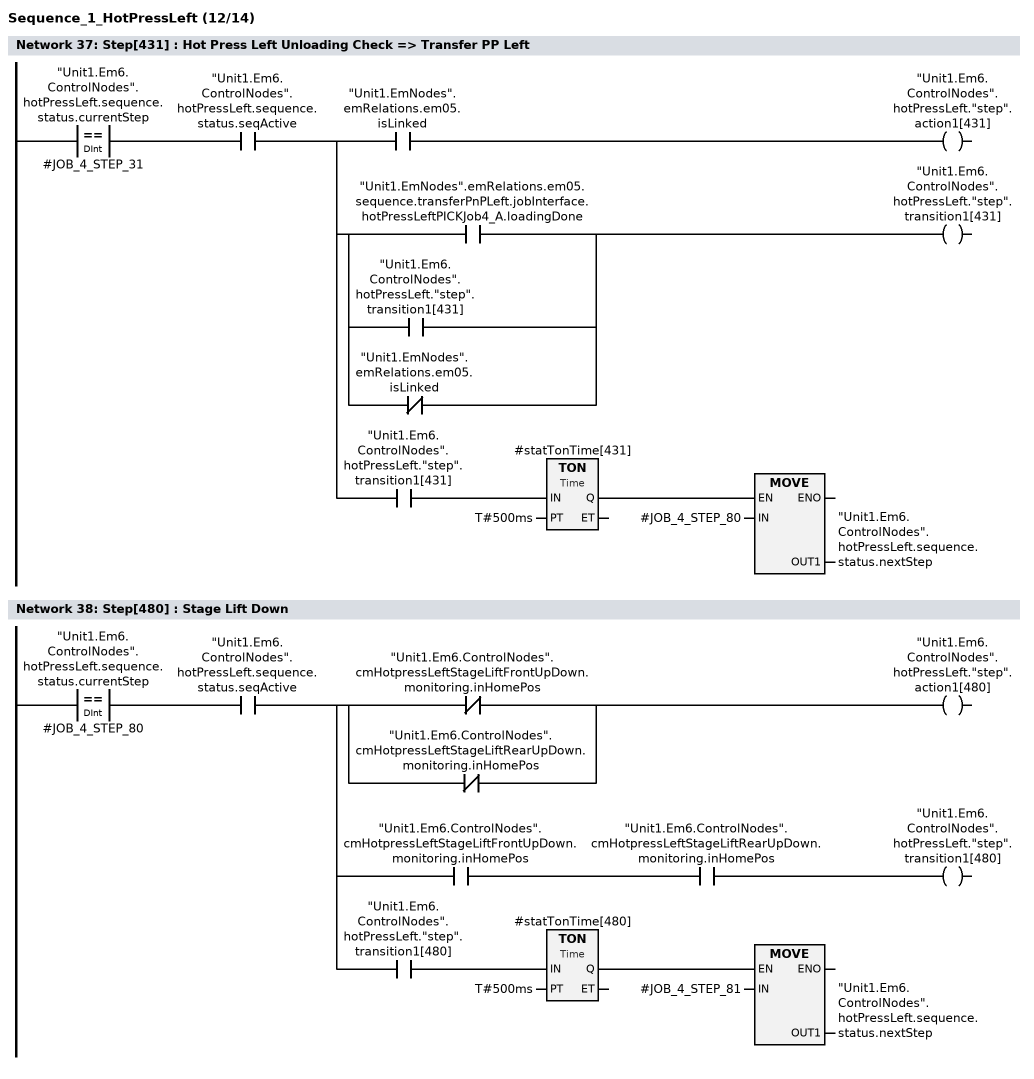
   RUNG wire#powerrail
      { S7_Templates := "SrcType := DInt" } EQ_Contact(in1 := "Unit1.Em6.ControlNodes".hotPressLeft.sequence.status.currentStep, in2 := #JOB_4_STEP_31)
      Contact( "Unit1.Em6.ControlNodes".hotPressLeft.sequence.status.seqActive )
      wire#w1
      Contact( "Unit1.EmNodes".emRelations.em05.isLinked )
      Coil( "Unit1.Em6.ControlNodes".hotPressLeft."step".action1[431] )
   END_RUNG
   RUNG wire#w1
      Contact( "Unit1.EmNodes".emRelations.em05.sequence.transferPnPLeft.jobInterface.hotPressLeftPICKJob4_A.loadingDone )
      wire#w2
      Coil( "Unit1.Em6.ControlNodes".hotPressLeft."step".transition1[431] )
   END_RUNG
   RUNG wire#w1
      Contact( "Unit1.Em6.ControlNodes".hotPressLeft."step".transition1[431] )
   END_RUNG wire#w2
   RUNG wire#w1
      I_Contact( "Unit1.EmNodes".emRelations.em05.isLinked )
   END_RUNG wire#w2
   RUNG wire#w1
      Contact( "Unit1.Em6.ControlNodes".hotPressLeft."step".transition1[431] )
      { S7_Templates := "time_type := Time" } #statTonTime[431].TON(pt := T#500ms, et =>)
      Move(in := #JOB_4_STEP_80, out1 => "Unit1.Em6.ControlNodes".hotPressLeft.sequence.status.nextStep)
   END_RUNG
   // the same network as SCL:
   #_w1 := ("Unit1.Em6.ControlNodes".hotPressLeft.sequence.status.currentStep = #JOB_4_STEP_31) AND "Unit1.Em6.ControlNodes".hotPressLeft.sequence.status.seqActive;
   "Unit1.Em6.ControlNodes".hotPressLeft."step".action1[431] := #_w1 AND "Unit1.EmNodes".emRelations.em05.isLinked;
   "Unit1.Em6.ControlNodes".hotPressLeft."step".transition1[431] := #_w1 AND ("Unit1.EmNodes".emRelations.em05.sequence.transferPnPLeft.jobInterface.hotPressLeftPICKJob4_A.loadingDone OR "Unit1.Em6.ControlNodes".hotPressLeft."step".transition1[431] OR NOT "Unit1.EmNodes".emRelations.em05.isLinked);
   #statTonTime[431].TON(IN := #_w1 AND "Unit1.Em6.ControlNodes".hotPressLeft."step".transition1[431],
                         PT := T#500ms);
   IF #statTonTime[431].Q THEN
       "Unit1.Em6.ControlNodes".hotPressLeft.sequence.status.nextStep := #JOB_4_STEP_80;
   END_IF;
END_REGION

REGION Network 38: Step[480] : Stage Lift Down
   RUNG wire#powerrail
      { S7_Templates := "SrcType := DInt" } EQ_Contact(in1 := "Unit1.Em6.ControlNodes".hotPressLeft.sequence.status.currentStep, in2 := #JOB_4_STEP_80)
      Contact( "Unit1.Em6.ControlNodes".hotPressLeft.sequence.status.seqActive )
      wire#w1
      I_Contact( "Unit1.Em6.ControlNodes".cmHotpressLeftStageLiftFrontUpDown.monitoring.inHomePos )
      wire#w2
      Coil( "Unit1.Em6.ControlNodes".hotPressLeft."step".action1[480] )
   END_RUNG
   RUNG wire#w1
      I_Contact( "Unit1.Em6.ControlNodes".cmHotpressLeftStageLiftRearUpDown.monitoring.inHomePos )
   END_RUNG wire#w2
   RUNG wire#w1
      Contact( "Unit1.Em6.ControlNodes".cmHotpressLeftStageLiftFrontUpDown.monitoring.inHomePos )
      Contact( "Unit1.Em6.ControlNodes".cmHotpressLeftStageLiftRearUpDown.monitoring.inHomePos )
      Coil( "Unit1.Em6.ControlNodes".hotPressLeft."step".transition1[480] )
   END_RUNG
   RUNG wire#w1
      Contact( "Unit1.Em6.ControlNodes".hotPressLeft."step".transition1[480] )
      { S7_Templates := "time_type := Time" } #statTonTime[480].TON(pt := T#500ms, et =>)
      Move(in := #JOB_4_STEP_81, out1 => "Unit1.Em6.ControlNodes".hotPressLeft.sequence.status.nextStep)
   END_RUNG
   // the same network as SCL:
   #_w1 := ("Unit1.Em6.ControlNodes".hotPressLeft.sequence.status.currentStep = #JOB_4_STEP_80) AND "Unit1.Em6.ControlNodes".hotPressLeft.sequence.status.seqActive;
   "Unit1.Em6.ControlNodes".hotPressLeft."step".action1[480] := #_w1 AND (NOT "Unit1.Em6.ControlNodes".cmHotpressLeftStageLiftFrontUpDown.monitoring.inHomePos OR NOT "Unit1.Em6.ControlNodes".cmHotpressLeftStageLiftRearUpDown.monitoring.inHomePos);
   "Unit1.Em6.ControlNodes".hotPressLeft."step".transition1[480] := #_w1 AND "Unit1.Em6.ControlNodes".cmHotpressLeftStageLiftFrontUpDown.monitoring.inHomePos AND "Unit1.Em6.ControlNodes".cmHotpressLeftStageLiftRearUpDown.monitoring.inHomePos;
   #statTonTime[480].TON(IN := #_w1 AND "Unit1.Em6.ControlNodes".hotPressLeft."step".transition1[480],
                         PT := T#500ms);
   IF #statTonTime[480].Q THEN
       "Unit1.Em6.ControlNodes".hotPressLeft.sequence.status.nextStep := #JOB_4_STEP_81;
   END_IF;
END_REGION

REGION Network 39: Step[481] : Spare
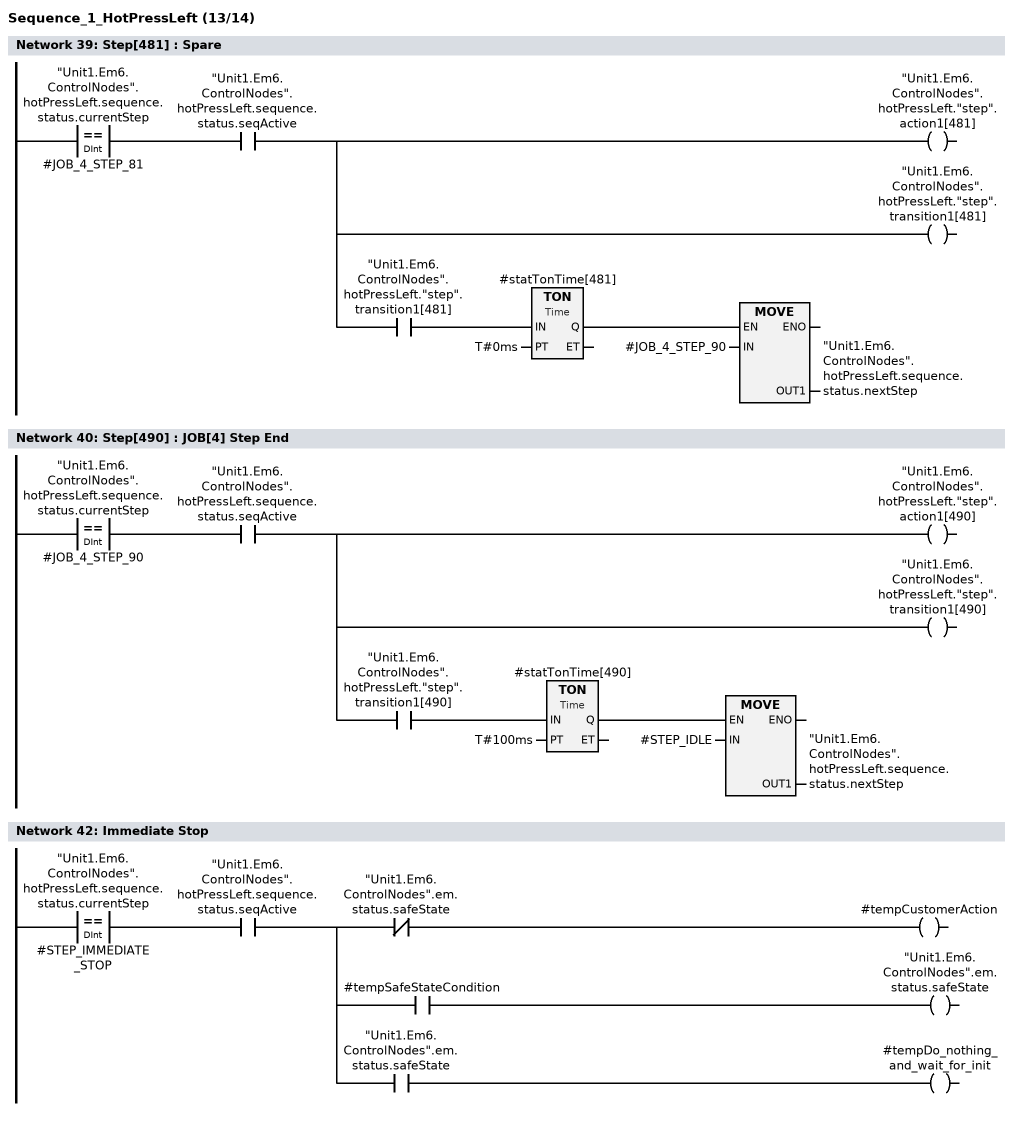
   RUNG wire#powerrail
      { S7_Templates := "SrcType := DInt" } EQ_Contact(in1 := "Unit1.Em6.ControlNodes".hotPressLeft.sequence.status.currentStep, in2 := #JOB_4_STEP_81)
      Contact( "Unit1.Em6.ControlNodes".hotPressLeft.sequence.status.seqActive )
      wire#w1
      Coil( "Unit1.Em6.ControlNodes".hotPressLeft."step".action1[481] )
   END_RUNG
   RUNG wire#w1
      Coil( "Unit1.Em6.ControlNodes".hotPressLeft."step".transition1[481] )
   END_RUNG
   RUNG wire#w1
      Contact( "Unit1.Em6.ControlNodes".hotPressLeft."step".transition1[481] )
      { S7_Templates := "time_type := Time" } #statTonTime[481].TON(pt := T#0ms, et =>)
      Move(in := #JOB_4_STEP_90, out1 => "Unit1.Em6.ControlNodes".hotPressLeft.sequence.status.nextStep)
   END_RUNG
   // the same network as SCL:
   "Unit1.Em6.ControlNodes".hotPressLeft."step".action1[481] := ("Unit1.Em6.ControlNodes".hotPressLeft.sequence.status.currentStep = #JOB_4_STEP_81) AND "Unit1.Em6.ControlNodes".hotPressLeft.sequence.status.seqActive;
   "Unit1.Em6.ControlNodes".hotPressLeft."step".transition1[481] := ("Unit1.Em6.ControlNodes".hotPressLeft.sequence.status.currentStep = #JOB_4_STEP_81) AND "Unit1.Em6.ControlNodes".hotPressLeft.sequence.status.seqActive;
   #statTonTime[481].TON(IN := ("Unit1.Em6.ControlNodes".hotPressLeft.sequence.status.currentStep = #JOB_4_STEP_81) AND "Unit1.Em6.ControlNodes".hotPressLeft.sequence.status.seqActive AND "Unit1.Em6.ControlNodes".hotPressLeft."step".transition1[481],
                         PT := T#0ms);
   IF #statTonTime[481].Q THEN
       "Unit1.Em6.ControlNodes".hotPressLeft.sequence.status.nextStep := #JOB_4_STEP_90;
   END_IF;
END_REGION

REGION Network 40: Step[490] : JOB[4] Step End
   RUNG wire#powerrail
      { S7_Templates := "SrcType := DInt" } EQ_Contact(in1 := "Unit1.Em6.ControlNodes".hotPressLeft.sequence.status.currentStep, in2 := #JOB_4_STEP_90)
      Contact( "Unit1.Em6.ControlNodes".hotPressLeft.sequence.status.seqActive )
      wire#w1
      Coil( "Unit1.Em6.ControlNodes".hotPressLeft."step".action1[490] )
   END_RUNG
   RUNG wire#w1
      Coil( "Unit1.Em6.ControlNodes".hotPressLeft."step".transition1[490] )
   END_RUNG
   RUNG wire#w1
      Contact( "Unit1.Em6.ControlNodes".hotPressLeft."step".transition1[490] )
      { S7_Templates := "time_type := Time" } #statTonTime[490].TON(pt := T#100ms, et =>)
      Move(in := #STEP_IDLE, out1 => "Unit1.Em6.ControlNodes".hotPressLeft.sequence.status.nextStep)
   END_RUNG
   // the same network as SCL:
   "Unit1.Em6.ControlNodes".hotPressLeft."step".action1[490] := ("Unit1.Em6.ControlNodes".hotPressLeft.sequence.status.currentStep = #JOB_4_STEP_90) AND "Unit1.Em6.ControlNodes".hotPressLeft.sequence.status.seqActive;
   "Unit1.Em6.ControlNodes".hotPressLeft."step".transition1[490] := ("Unit1.Em6.ControlNodes".hotPressLeft.sequence.status.currentStep = #JOB_4_STEP_90) AND "Unit1.Em6.ControlNodes".hotPressLeft.sequence.status.seqActive;
   #statTonTime[490].TON(IN := ("Unit1.Em6.ControlNodes".hotPressLeft.sequence.status.currentStep = #JOB_4_STEP_90) AND "Unit1.Em6.ControlNodes".hotPressLeft.sequence.status.seqActive AND "Unit1.Em6.ControlNodes".hotPressLeft."step".transition1[490],
                         PT := T#100ms);
   IF #statTonTime[490].Q THEN
       "Unit1.Em6.ControlNodes".hotPressLeft.sequence.status.nextStep := #STEP_IDLE;
   END_IF;
END_REGION

REGION Network 41: ******************** IMMEDIATE STOP *********************
END_REGION

REGION Network 42: Immediate Stop
   RUNG wire#powerrail
      { S7_Templates := "SrcType := DInt" } EQ_Contact(in1 := "Unit1.Em6.ControlNodes".hotPressLeft.sequence.status.currentStep, in2 := #STEP_IMMEDIATE_STOP)
      Contact( "Unit1.Em6.ControlNodes".hotPressLeft.sequence.status.seqActive )
      wire#w1
      I_Contact( "Unit1.Em6.ControlNodes".em.status.safeState )
      Coil( #tempCustomerAction )
   END_RUNG
   RUNG wire#w1
      Contact( #tempSafeStateCondition )
      Coil( "Unit1.Em6.ControlNodes".em.status.safeState )
   END_RUNG
   RUNG wire#w1
      Contact( "Unit1.Em6.ControlNodes".em.status.safeState )
      Coil( #tempDo_nothing_and_wait_for_init )
   END_RUNG
   // the same network as SCL:
   #_w1 := ("Unit1.Em6.ControlNodes".hotPressLeft.sequence.status.currentStep = #STEP_IMMEDIATE_STOP) AND "Unit1.Em6.ControlNodes".hotPressLeft.sequence.status.seqActive;
   #tempCustomerAction := #_w1 AND NOT "Unit1.Em6.ControlNodes".em.status.safeState;
   "Unit1.Em6.ControlNodes".em.status.safeState := #_w1 AND #tempSafeStateCondition;
   #tempDo_nothing_and_wait_for_init := #_w1 AND "Unit1.Em6.ControlNodes".em.status.safeState;
END_REGION

REGION Network 43: ********************** STATUS **************************
END_REGION

REGION Network 44: Sequence Status
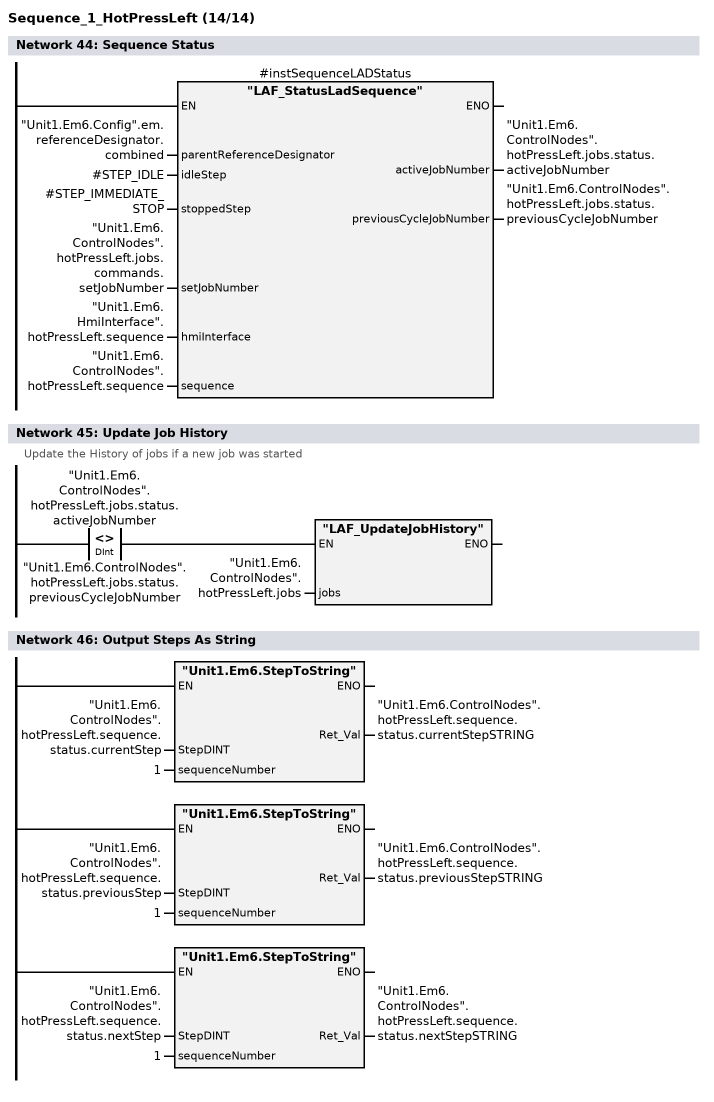
   RUNG wire#powerrail
      #instSequenceLADStatus(parentReferenceDesignator := "Unit1.Em6.Config".em.referenceDesignator.combined, idleStep := #STEP_IDLE, stoppedStep := #STEP_IMMEDIATE_STOP, setJobNumber := "Unit1.Em6.ControlNodes".hotPressLeft.jobs.commands.setJobNumber, hmiInterface := "Unit1.Em6.HmiInterface".hotPressLeft.sequence, sequence := "Unit1.Em6.ControlNodes".hotPressLeft.sequence, activeJobNumber => "Unit1.Em6.ControlNodes".hotPressLeft.jobs.status.activeJobNumber, previousCycleJobNumber => "Unit1.Em6.ControlNodes".hotPressLeft.jobs.status.previousCycleJobNumber)
   END_RUNG
   // the same network as SCL:
   #instSequenceLADStatus(parentReferenceDesignator := "Unit1.Em6.Config".em.referenceDesignator.combined,   // "LAF_StatusLadSequence"
                          idleStep := #STEP_IDLE,
                          stoppedStep := #STEP_IMMEDIATE_STOP,
                          setJobNumber := "Unit1.Em6.ControlNodes".hotPressLeft.jobs.commands.setJobNumber,
                          hmiInterface := "Unit1.Em6.HmiInterface".hotPressLeft.sequence,
                          sequence := "Unit1.Em6.ControlNodes".hotPressLeft.sequence,
                          activeJobNumber => "Unit1.Em6.ControlNodes".hotPressLeft.jobs.status.activeJobNumber,
                          previousCycleJobNumber => "Unit1.Em6.ControlNodes".hotPressLeft.jobs.status.previousCycleJobNumber);
END_REGION

REGION Network 45: Update Job History
   // Update the History of jobs if a new job was started
   RUNG wire#powerrail
      { S7_Templates := "SrcType := DInt" } NE_Contact(in1 := "Unit1.Em6.ControlNodes".hotPressLeft.jobs.status.activeJobNumber, in2 := "Unit1.Em6.ControlNodes".hotPressLeft.jobs.status.previousCycleJobNumber)
      "LAF_UpdateJobHistory"(jobs := "Unit1.Em6.ControlNodes".hotPressLeft.jobs)
   END_RUNG
   // the same network as SCL:
   IF "Unit1.Em6.ControlNodes".hotPressLeft.jobs.status.activeJobNumber <> "Unit1.Em6.ControlNodes".hotPressLeft.jobs.status.previousCycleJobNumber THEN
       "LAF_UpdateJobHistory"(jobs := "Unit1.Em6.ControlNodes".hotPressLeft.jobs);
   END_IF;
END_REGION

REGION Network 46: Output Steps As String
   RUNG wire#powerrail
      "Unit1.Em6.StepToString"(StepDINT := "Unit1.Em6.ControlNodes".hotPressLeft.sequence.status.currentStep, sequenceNumber := 1, Ret_Val => "Unit1.Em6.ControlNodes".hotPressLeft.sequence.status.currentStepSTRING)
   END_RUNG
   RUNG wire#powerrail
      "Unit1.Em6.StepToString"(StepDINT := "Unit1.Em6.ControlNodes".hotPressLeft.sequence.status.previousStep, sequenceNumber := 1, Ret_Val => "Unit1.Em6.ControlNodes".hotPressLeft.sequence.status.previousStepSTRING)
   END_RUNG
   RUNG wire#powerrail
      "Unit1.Em6.StepToString"(StepDINT := "Unit1.Em6.ControlNodes".hotPressLeft.sequence.status.nextStep, sequenceNumber := 1, Ret_Val => "Unit1.Em6.ControlNodes".hotPressLeft.sequence.status.nextStepSTRING)
   END_RUNG
   // the same network as SCL:
   "Unit1.Em6.ControlNodes".hotPressLeft.sequence.status.currentStepSTRING := "Unit1.Em6.StepToString"(StepDINT := "Unit1.Em6.ControlNodes".hotPressLeft.sequence.status.currentStep,
                           sequenceNumber := 1);
   "Unit1.Em6.ControlNodes".hotPressLeft.sequence.status.previousStepSTRING := "Unit1.Em6.StepToString"(StepDINT := "Unit1.Em6.ControlNodes".hotPressLeft.sequence.status.previousStep,
                           sequenceNumber := 1);
   "Unit1.Em6.ControlNodes".hotPressLeft.sequence.status.nextStepSTRING := "Unit1.Em6.StepToString"(StepDINT := "Unit1.Em6.ControlNodes".hotPressLeft.sequence.status.nextStep,
                           sequenceNumber := 1);
END_REGION
END_FUNCTION_BLOCK
